					FOR CallRTBFL := 1 TO iRecipeBlockQty DO
						IF CallRTBFL > 0 AND CallRTBFL <= iRecipeBlockQty THEN
						AR2SiCalledRecipeTimeBlockNoCallArmTime[CallRTBFL, 1] :=	 AR3SiRecipeTimeBlockMemoryNoCallArmTime[iAutoModeCallRecipeTimeBlock_ProductRecipeNo, CallRTBFL, 1];
						AR2SiCalledRecipeTimeBlockNoCallArmTime[CallRTBFL, 2] :=	 AR3SiRecipeTimeBlockMemoryNoCallArmTime[iAutoModeCallRecipeTimeBlock_ProductRecipeNo, CallRTBFL, 2];
						AR2SiCalledRecipeTimeBlockNoCallArmTime[CallRTBFL, 3] :=	 AR3SiRecipeTimeBlockMemoryNoCallArmTime[iAutoModeCallRecipeTimeBlock_ProductRecipeNo, CallRTBFL, 3];
						AR2SiCalledRecipeTimeBlockNoCallArmTime[CallRTBFL, 4] :=	 AR3SiRecipeTimeBlockMemoryNoCallArmTime[iAutoModeCallRecipeTimeBlock_ProductRecipeNo, CallRTBFL, 4];
						AR2SiCalledRecipeTimeBlockNoCallArmTime[CallRTBFL, 5] :=	 AR3SiRecipeTimeBlockMemoryNoCallArmTime[iAutoModeCallRecipeTimeBlock_ProductRecipeNo, CallRTBFL, 5];
						AR2SiCalledRecipeTimeBlockNoCallArmTime[CallRTBFL, 6] :=	 AR3SiRecipeTimeBlockMemoryNoCallArmTime[iAutoModeCallRecipeTimeBlock_ProductRecipeNo, CallRTBFL, 6];
						AR2SiCalledRecipeTimeBlockNoCallArmTime[CallRTBFL, 7] :=	 AR3SiRecipeTimeBlockMemoryNoCallArmTime[iAutoModeCallRecipeTimeBlock_ProductRecipeNo, CallRTBFL, 7];
						AR2SiCalledRecipeTimeBlockNoCallArmTime[CallRTBFL, 8] :=	 AR3SiRecipeTimeBlockMemoryNoCallArmTime[iAutoModeCallRecipeTimeBlock_ProductRecipeNo, CallRTBFL, 8];
						AR2SiCalledRecipeTimeBlockNoCallArmTime[CallRTBFL, 9] :=	 AR3SiRecipeTimeBlockMemoryNoCallArmTime[iAutoModeCallRecipeTimeBlock_ProductRecipeNo, CallRTBFL, 9];
						END_IF
					END_FOR


				END_IF


				IF AR3SiRecipeTimeBlockMemoryWithCallArmTime[iAutoModeCallRecipeTimeBlock_ProductRecipeNo, 1, 3] <> 0 THEN
				CallRTBFL := 1;

					FOR CallRTBFL := 1 TO iRecipeBlockQty DO
						IF CallRTBFL > 0 AND CallRTBFL <= iRecipeBlockQty THEN
						AR2SiCalledRecipeTimeBlockWithCallArmTime[CallRTBFL, 1] :=	 AR3SiRecipeTimeBlockMemoryWithCallArmTime[iAutoModeCallRecipeTimeBlock_ProductRecipeNo, CallRTBFL, 1];
						AR2SiCalledRecipeTimeBlockWithCallArmTime[CallRTBFL, 2] :=	 AR3SiRecipeTimeBlockMemoryWithCallArmTime[iAutoModeCallRecipeTimeBlock_ProductRecipeNo, CallRTBFL, 2];
						AR2SiCalledRecipeTimeBlockWithCallArmTime[CallRTBFL, 3] :=	 AR3SiRecipeTimeBlockMemoryWithCallArmTime[iAutoModeCallRecipeTimeBlock_ProductRecipeNo, CallRTBFL, 3];
						AR2SiCalledRecipeTimeBlockWithCallArmTime[CallRTBFL, 4] :=	 AR3SiRecipeTimeBlockMemoryWithCallArmTime[iAutoModeCallRecipeTimeBlock_ProductRecipeNo, CallRTBFL, 4];
						AR2SiCalledRecipeTimeBlockWithCallArmTime[CallRTBFL, 5] :=	 AR3SiRecipeTimeBlockMemoryWithCallArmTime[iAutoModeCallRecipeTimeBlock_ProductRecipeNo, CallRTBFL, 5];
						AR2SiCalledRecipeTimeBlockWithCallArmTime[CallRTBFL, 6] :=	 AR3SiRecipeTimeBlockMemoryWithCallArmTime[iAutoModeCallRecipeTimeBlock_ProductRecipeNo, CallRTBFL, 6];
						AR2SiCalledRecipeTimeBlockWithCallArmTime[CallRTBFL, 7] :=	 AR3SiRecipeTimeBlockMemoryWithCallArmTime[iAutoModeCallRecipeTimeBlock_ProductRecipeNo, CallRTBFL, 7];
						AR2SiCalledRecipeTimeBlockWithCallArmTime[CallRTBFL, 8] :=	 AR3SiRecipeTimeBlockMemoryWithCallArmTime[iAutoModeCallRecipeTimeBlock_ProductRecipeNo, CallRTBFL, 8];
						AR2SiCalledRecipeTimeBlockWithCallArmTime[CallRTBFL, 9] :=	 AR3SiRecipeTimeBlockMemoryWithCallArmTime[iAutoModeCallRecipeTimeBlock_ProductRecipeNo, CallRTBFL, 9];
						END_IF
					END_FOR
			
			
				END_IF

			ELSE
			bInvalidCallRecipeTimeBlockNo := TRUE;
			END_IF

			IF AR2SiCalledRecipeTimeBlockWithCallArmTime [1,3] <> 0 THEN
			bCallRTB_NoTrackerInfo := FALSE;
			bCallRTB_CallOK := TRUE;
			END_IF

(*SimulatorMode Call*)
ELSIF bSimulatorModeEn
AND NOT bMasterTimeBlockScanningEn
AND NOT tProductRecipeChangesFound.Q
AND NOT  bScanningEN
AND iSimulatorModeCallRecipeTimeBlock_ProductRecipeNo >0
(*AND ARbProductRecipeTimeBlockAvailable[iSimulatorModeCallRecipeTimeBlock_ProductRecipeNo]
AND AR2SiCalledRecipeTimeBlockNoCallArmTime[1, 3] = 0*)
THEN

			IF iSimulatorModeCallRecipeTimeBlock_ProductRecipeNo >0 THEN
			AR2SiCalledRecipeTimeBlockNoCallArmTime := AR2SiCalledRecipeTimeBlockNoCallArmTimeEmpty;
			AR2SiCalledRecipeTimeBlockWithCallArmTime := AR2SiCalledRecipeTimeBlockWithCallArmTimeEmpty;
			bInvalidCallRecipeTimeBlockNo := FALSE;

				IF AR3SiRecipeTimeBlockMemoryNoCallArmTime[iSimulatorModeCallRecipeTimeBlock_ProductRecipeNo, 1, 3] <> 0 THEN
				CallRTBFL := 1;

					FOR CallRTBFL := 1 TO iRecipeBlockQty DO
						IF CallRTBFL > 0 AND CallRTBFL <= iRecipeBlockQty THEN
						AR2SiCalledRecipeTimeBlockNoCallArmTime[CallRTBFL, 1] :=	 AR3SiRecipeTimeBlockMemoryNoCallArmTime[iSimulatorModeCallRecipeTimeBlock_ProductRecipeNo, CallRTBFL, 1];
						AR2SiCalledRecipeTimeBlockNoCallArmTime[CallRTBFL, 2] :=	 AR3SiRecipeTimeBlockMemoryNoCallArmTime[iSimulatorModeCallRecipeTimeBlock_ProductRecipeNo, CallRTBFL, 2];
						AR2SiCalledRecipeTimeBlockNoCallArmTime[CallRTBFL, 3] :=	 AR3SiRecipeTimeBlockMemoryNoCallArmTime[iSimulatorModeCallRecipeTimeBlock_ProductRecipeNo, CallRTBFL, 3];
						AR2SiCalledRecipeTimeBlockNoCallArmTime[CallRTBFL, 4] :=	 AR3SiRecipeTimeBlockMemoryNoCallArmTime[iSimulatorModeCallRecipeTimeBlock_ProductRecipeNo, CallRTBFL, 4];
						AR2SiCalledRecipeTimeBlockNoCallArmTime[CallRTBFL, 5] :=	 AR3SiRecipeTimeBlockMemoryNoCallArmTime[iSimulatorModeCallRecipeTimeBlock_ProductRecipeNo, CallRTBFL, 5];
						AR2SiCalledRecipeTimeBlockNoCallArmTime[CallRTBFL, 6] :=	 AR3SiRecipeTimeBlockMemoryNoCallArmTime[iSimulatorModeCallRecipeTimeBlock_ProductRecipeNo, CallRTBFL, 6];
						AR2SiCalledRecipeTimeBlockNoCallArmTime[CallRTBFL, 7] :=	 AR3SiRecipeTimeBlockMemoryNoCallArmTime[iSimulatorModeCallRecipeTimeBlock_ProductRecipeNo, CallRTBFL, 7];
						AR2SiCalledRecipeTimeBlockNoCallArmTime[CallRTBFL, 8] :=	 AR3SiRecipeTimeBlockMemoryNoCallArmTime[iSimulatorModeCallRecipeTimeBlock_ProductRecipeNo, CallRTBFL, 8];
						AR2SiCalledRecipeTimeBlockNoCallArmTime[CallRTBFL, 9] :=	 AR3SiRecipeTimeBlockMemoryNoCallArmTime[iSimulatorModeCallRecipeTimeBlock_ProductRecipeNo, CallRTBFL, 9];
						END_IF
					END_FOR
			
			
				END_IF


				IF AR3SiRecipeTimeBlockMemoryWithCallArmTime[iSimulatorModeCallRecipeTimeBlock_ProductRecipeNo, 1, 3] <> 0 THEN
				CallRTBFL := 1;
			
					FOR CallRTBFL := 1 TO iRecipeBlockQty DO
						IF CallRTBFL > 0 AND CallRTBFL <= iRecipeBlockQty THEN
						AR2SiCalledRecipeTimeBlockWithCallArmTime[CallRTBFL, 1] :=	 AR3SiRecipeTimeBlockMemoryWithCallArmTime[iSimulatorModeCallRecipeTimeBlock_ProductRecipeNo, CallRTBFL, 1];
						AR2SiCalledRecipeTimeBlockWithCallArmTime[CallRTBFL, 2] :=	 AR3SiRecipeTimeBlockMemoryWithCallArmTime[iSimulatorModeCallRecipeTimeBlock_ProductRecipeNo, CallRTBFL, 2];
						AR2SiCalledRecipeTimeBlockWithCallArmTime[CallRTBFL, 3] :=	 AR3SiRecipeTimeBlockMemoryWithCallArmTime[iSimulatorModeCallRecipeTimeBlock_ProductRecipeNo, CallRTBFL, 3];
						AR2SiCalledRecipeTimeBlockWithCallArmTime[CallRTBFL, 4] :=	 AR3SiRecipeTimeBlockMemoryWithCallArmTime[iSimulatorModeCallRecipeTimeBlock_ProductRecipeNo, CallRTBFL, 4];
						AR2SiCalledRecipeTimeBlockWithCallArmTime[CallRTBFL, 5] :=	 AR3SiRecipeTimeBlockMemoryWithCallArmTime[iSimulatorModeCallRecipeTimeBlock_ProductRecipeNo, CallRTBFL, 5];
						AR2SiCalledRecipeTimeBlockWithCallArmTime[CallRTBFL, 6] :=	 AR3SiRecipeTimeBlockMemoryWithCallArmTime[iSimulatorModeCallRecipeTimeBlock_ProductRecipeNo, CallRTBFL, 6];
						AR2SiCalledRecipeTimeBlockWithCallArmTime[CallRTBFL, 7] :=	 AR3SiRecipeTimeBlockMemoryWithCallArmTime[iSimulatorModeCallRecipeTimeBlock_ProductRecipeNo, CallRTBFL, 7];
						AR2SiCalledRecipeTimeBlockWithCallArmTime[CallRTBFL, 8] :=	 AR3SiRecipeTimeBlockMemoryWithCallArmTime[iSimulatorModeCallRecipeTimeBlock_ProductRecipeNo, CallRTBFL, 8];
						AR2SiCalledRecipeTimeBlockWithCallArmTime[CallRTBFL, 9] :=	 AR3SiRecipeTimeBlockMemoryWithCallArmTime[iSimulatorModeCallRecipeTimeBlock_ProductRecipeNo, CallRTBFL, 9];
						END_IF
					END_FOR

			
				END_IF

			ELSE
			bInvalidCallRecipeTimeBlockNo := TRUE;
			END_IF


			IF AR2SiCalledRecipeTimeBlockWithCallArmTime [1,3] <> 0 THEN
			bCallRTB_NoTrackerInfo := FALSE;
			bCallRTB_CallOK := TRUE;
			END_IF


END_IF



(*Check Product Recipe Time Block Availibility *)
iCheckPRTBFL := 1;

	FOR iCheckPRTBFL := 1 TO iProductRecipeArrayQty DO
		IF iCheckPRTBFL >= 1 AND iCheckPRTBFL <= iProductRecipeArrayQty THEN

			IF  AR3SiRecipeTimeBlockMemoryNoCallArmTime[iCheckPRTBFL, 1, 3] > 0 THEN
			ARbProductRecipeTimeBlockAvailable[iCheckPRTBFL ] := TRUE;
			ELSE
			ARbProductRecipeTimeBlockAvailable[iCheckPRTBFL ] := FALSE;
			END_IF

		END_IF
	END_FOR

ACTION XML_ImportExport:
(* XML Import Export Control *)
(*	ARiSubAction					: ARRAY [1..10] OF INT; (* 0-Idle, 1-Import, 2-Export, 3-Clear/Delete 8-Done *)*)

	IF 		ARiSubAction[2] = 1 THEN (*Write from Buffer to Actual Memory*)

				CallRTBFL := 1;

					FOR CallRTBFL := 1 TO iRecipeBlockQty DO
						IF CallRTBFL > 0 AND CallRTBFL <= iRecipeBlockQty THEN
						AR3SiRecipeTimeBlockMemoryNoCallArmTime[iXMLRecipeNo, CallRTBFL, 1] :=	 DSV3XML_Recipe.AR2SiRecipeTimeBlockNoCallArmTime[CallRTBFL, 1];
						AR3SiRecipeTimeBlockMemoryNoCallArmTime[iXMLRecipeNo, CallRTBFL, 2] :=	 DSV3XML_Recipe.AR2SiRecipeTimeBlockNoCallArmTime[CallRTBFL, 2];
						AR3SiRecipeTimeBlockMemoryNoCallArmTime[iXMLRecipeNo, CallRTBFL, 3] :=	 DSV3XML_Recipe.AR2SiRecipeTimeBlockNoCallArmTime[CallRTBFL, 3];
						AR3SiRecipeTimeBlockMemoryNoCallArmTime[iXMLRecipeNo, CallRTBFL, 4] :=	 DSV3XML_Recipe.AR2SiRecipeTimeBlockNoCallArmTime[CallRTBFL, 4];
						AR3SiRecipeTimeBlockMemoryNoCallArmTime[iXMLRecipeNo, CallRTBFL, 5] :=	 DSV3XML_Recipe.AR2SiRecipeTimeBlockNoCallArmTime[CallRTBFL, 5];
						AR3SiRecipeTimeBlockMemoryNoCallArmTime[iXMLRecipeNo, CallRTBFL, 6] :=	 DSV3XML_Recipe.AR2SiRecipeTimeBlockNoCallArmTime[CallRTBFL, 6];
						AR3SiRecipeTimeBlockMemoryNoCallArmTime[iXMLRecipeNo, CallRTBFL, 7] :=	 DSV3XML_Recipe.AR2SiRecipeTimeBlockNoCallArmTime[CallRTBFL, 7];
						AR3SiRecipeTimeBlockMemoryNoCallArmTime[iXMLRecipeNo, CallRTBFL, 8] :=	 DSV3XML_Recipe.AR2SiRecipeTimeBlockNoCallArmTime[CallRTBFL, 8];
						AR3SiRecipeTimeBlockMemoryNoCallArmTime[iXMLRecipeNo, CallRTBFL, 9] :=	 DSV3XML_Recipe.AR2SiRecipeTimeBlockNoCallArmTime[CallRTBFL, 9];

						AR3SiRecipeTimeBlockMemoryWithCallArmTime[iXMLRecipeNo, CallRTBFL, 1] :=	 DSV3XML_Recipe.AR2SiRecipeTimeBlockWithCallArmTime[CallRTBFL, 1];
						AR3SiRecipeTimeBlockMemoryWithCallArmTime[iXMLRecipeNo, CallRTBFL, 2] :=	 DSV3XML_Recipe.AR2SiRecipeTimeBlockWithCallArmTime[CallRTBFL, 2];
						AR3SiRecipeTimeBlockMemoryWithCallArmTime[iXMLRecipeNo, CallRTBFL, 3] :=	 DSV3XML_Recipe.AR2SiRecipeTimeBlockWithCallArmTime[CallRTBFL, 3];
						AR3SiRecipeTimeBlockMemoryWithCallArmTime[iXMLRecipeNo, CallRTBFL, 4] :=	 DSV3XML_Recipe.AR2SiRecipeTimeBlockWithCallArmTime[CallRTBFL, 4];
						AR3SiRecipeTimeBlockMemoryWithCallArmTime[iXMLRecipeNo, CallRTBFL, 5] :=	 DSV3XML_Recipe.AR2SiRecipeTimeBlockWithCallArmTime[CallRTBFL, 5];
						AR3SiRecipeTimeBlockMemoryWithCallArmTime[iXMLRecipeNo, CallRTBFL, 6] :=	 DSV3XML_Recipe.AR2SiRecipeTimeBlockWithCallArmTime[CallRTBFL, 6];
						AR3SiRecipeTimeBlockMemoryWithCallArmTime[iXMLRecipeNo, CallRTBFL, 7] :=	 DSV3XML_Recipe.AR2SiRecipeTimeBlockWithCallArmTime[CallRTBFL, 7];
						AR3SiRecipeTimeBlockMemoryWithCallArmTime[iXMLRecipeNo, CallRTBFL, 8] :=	 DSV3XML_Recipe.AR2SiRecipeTimeBlockWithCallArmTime[CallRTBFL, 8];
						AR3SiRecipeTimeBlockMemoryWithCallArmTime[iXMLRecipeNo, CallRTBFL, 9] :=	 DSV3XML_Recipe.AR2SiRecipeTimeBlockWithCallArmTime[CallRTBFL, 9];
						END_IF
					END_FOR

				ARbProductRecipeTimeBlockAvailable[iXMLRecipeNo] := DSV3XML_Recipe.bProductRecipeTimeBlockAvailable ;

				ARiSubAction[2] := 8;
(*				IF iHMIRecipeNo = iXMLRecipeNo THEN
					bRecipeLoadPb := TRUE;
				END_IF
*)
	ELSIF	ARiSubAction[2] = 2 THEN (*Read from Actual to Buffer Memory*)

				CallRTBFL := 1;

					FOR CallRTBFL := 1 TO iRecipeBlockQty DO
						IF CallRTBFL > 0 AND CallRTBFL <= iRecipeBlockQty THEN
						DSV3XML_Recipe.AR2SiRecipeTimeBlockNoCallArmTime[CallRTBFL, 1] :=	 AR3SiRecipeTimeBlockMemoryNoCallArmTime[iXMLRecipeNo, CallRTBFL, 1];
						DSV3XML_Recipe.AR2SiRecipeTimeBlockNoCallArmTime[CallRTBFL, 2] :=	 AR3SiRecipeTimeBlockMemoryNoCallArmTime[iXMLRecipeNo, CallRTBFL, 2];
						DSV3XML_Recipe.AR2SiRecipeTimeBlockNoCallArmTime[CallRTBFL, 3] :=	 AR3SiRecipeTimeBlockMemoryNoCallArmTime[iXMLRecipeNo, CallRTBFL, 3];
						DSV3XML_Recipe.AR2SiRecipeTimeBlockNoCallArmTime[CallRTBFL, 4] :=	 AR3SiRecipeTimeBlockMemoryNoCallArmTime[iXMLRecipeNo, CallRTBFL, 4];
						DSV3XML_Recipe.AR2SiRecipeTimeBlockNoCallArmTime[CallRTBFL, 5] :=	 AR3SiRecipeTimeBlockMemoryNoCallArmTime[iXMLRecipeNo, CallRTBFL, 5];
						DSV3XML_Recipe.AR2SiRecipeTimeBlockNoCallArmTime[CallRTBFL, 6] :=	 AR3SiRecipeTimeBlockMemoryNoCallArmTime[iXMLRecipeNo, CallRTBFL, 6];
						DSV3XML_Recipe.AR2SiRecipeTimeBlockNoCallArmTime[CallRTBFL, 7] :=	 AR3SiRecipeTimeBlockMemoryNoCallArmTime[iXMLRecipeNo, CallRTBFL, 7];
						DSV3XML_Recipe.AR2SiRecipeTimeBlockNoCallArmTime[CallRTBFL, 8] :=	 AR3SiRecipeTimeBlockMemoryNoCallArmTime[iXMLRecipeNo, CallRTBFL, 8];
						DSV3XML_Recipe.AR2SiRecipeTimeBlockNoCallArmTime[CallRTBFL, 9] :=	 AR3SiRecipeTimeBlockMemoryNoCallArmTime[iXMLRecipeNo, CallRTBFL, 9];

						DSV3XML_Recipe.AR2SiRecipeTimeBlockWithCallArmTime[CallRTBFL, 1] :=	 AR3SiRecipeTimeBlockMemoryWithCallArmTime[iXMLRecipeNo, CallRTBFL, 1];
						DSV3XML_Recipe.AR2SiRecipeTimeBlockWithCallArmTime[CallRTBFL, 2] :=	 AR3SiRecipeTimeBlockMemoryWithCallArmTime[iXMLRecipeNo, CallRTBFL, 2];
						DSV3XML_Recipe.AR2SiRecipeTimeBlockWithCallArmTime[CallRTBFL, 3] :=	 AR3SiRecipeTimeBlockMemoryWithCallArmTime[iXMLRecipeNo, CallRTBFL, 3];
						DSV3XML_Recipe.AR2SiRecipeTimeBlockWithCallArmTime[CallRTBFL, 4] :=	 AR3SiRecipeTimeBlockMemoryWithCallArmTime[iXMLRecipeNo, CallRTBFL, 4];
						DSV3XML_Recipe.AR2SiRecipeTimeBlockWithCallArmTime[CallRTBFL, 5] :=	 AR3SiRecipeTimeBlockMemoryWithCallArmTime[iXMLRecipeNo, CallRTBFL, 5];
						DSV3XML_Recipe.AR2SiRecipeTimeBlockWithCallArmTime[CallRTBFL, 6] :=	 AR3SiRecipeTimeBlockMemoryWithCallArmTime[iXMLRecipeNo, CallRTBFL, 6];
						DSV3XML_Recipe.AR2SiRecipeTimeBlockWithCallArmTime[CallRTBFL, 7] :=	 AR3SiRecipeTimeBlockMemoryWithCallArmTime[iXMLRecipeNo, CallRTBFL, 7];
						DSV3XML_Recipe.AR2SiRecipeTimeBlockWithCallArmTime[CallRTBFL, 8] :=	 AR3SiRecipeTimeBlockMemoryWithCallArmTime[iXMLRecipeNo, CallRTBFL, 8];
						DSV3XML_Recipe.AR2SiRecipeTimeBlockWithCallArmTime[CallRTBFL, 9] :=	 AR3SiRecipeTimeBlockMemoryWithCallArmTime[iXMLRecipeNo, CallRTBFL, 9];
						END_IF
					END_FOR

				DSV3XML_Recipe.bProductRecipeTimeBlockAvailable := ARbProductRecipeTimeBlockAvailable[iXMLRecipeNo];

				ARiSubAction[2] := 8;

	ELSIF	ARiSubAction[2] = 3 THEN (*DELETE Actual Memory*)

				AR3SiRecipeTimeBlockMemoryNoCallArmTime		:= AR3SiRecipeTimeBlockMemoryNoCallArmTime_Delete;
				AR3SiRecipeTimeBlockMemoryWithCallArmTime 		:= AR3SiRecipeTimeBlockMemoryWithCallArmTime_Delete;
				ARbProductRecipeTimeBlockAvailable 				:= ARbProductRecipeTimeBlockAvailable_Delete;

				ARiSubAction[2] := 8;
(*				IF iHMIRecipeNo = iXMLRecipeNo THEN
					bRecipeLoadPb := TRUE;
				END_IF
*)
	END_IF
END_ACTION

END_FUNCTION_BLOCK

// ---- FBs/B_JKS_NewFB_V3/UserCtrl/FB3_HmiTF1800_UserlevelManagement.TcPOU
FUNCTION_BLOCK FB3_HmiTF1800_UserlevelManagement
VAR_INPUT
	
	bLoginPB 					: BOOL;
	bLogoutPB 					: BOOL;
	iLoginNameId 				: REFERENCE TO INT; // The LoginName selection in HMI during User Login Pop-up Screen, the choosen user will translated as Array ID No and pass here.
	sPasswordField 				: REFERENCE TO STRING; // Similar to Var In/Out so that i can clear the password if login failed
	
	iUM_SelectedLoginNameId	 	: REFERENCE TO INT;		// User Management - Selected Login Name ID (Array No)

	sUM_CurrentPassword			: REFERENCE TO STRING;	// User Management - Current Password (For password change only)
	sUM_NewPassword				: REFERENCE TO STRING;	// User Management - New Password (For password change or new user registration)
	sUM_ConfirmPassword			: REFERENCE TO STRING;	// User Management - New Password (For password change or new user registration)

	sUM_NewUserLoginName		: REFERENCE TO STRING;	// User Management - New User Login Name
	sUM_NewUserGroupId			: REFERENCE TO INT;		// User Management - Select from UserGroupList

	sUM_NewUserOperatorIdentifier	: REFERENCE TO STRING;
	sUM_NewUserActorType			: REFERENCE TO eActor;
	sUM_NewUserLastName				: REFERENCE TO STRING;
	sUM_NewUserFirstName			: REFERENCE TO STRING;
//	sUM_NewUserGroupName			: REFERENCE TO WSTRING; // Generated by reference eto sUM_NewUserGroupId
	
	bUM_CreatePB				: BOOL;		// User Management - Button for New User creation
	bUM_EditPB					: BOOL;		// User Management - Button for Edit User
	bUM_DeletePB				: BOOL;		// User Management - Button for Delete User
	bUM_EnablePB				: BOOL; 	// to Enable selected User
	bUM_DisablePB				: BOOL; 	// to Temporary Disable selected User
	bUM_ConfirmPB				: BOOL;		// for Edit, Delete and Disable used. click to save
	bUM_ReturnPB				: BOOL;		// for Edit, Delete and Disable used, click to return without save.
		
END_VAR
VAR_OUTPUT
	dsHmiUserStatus_Active		: DS_HmiUserStatus;
	dsHmiUserStatus_Login		: DS_HmiUserStatus;
	dsHmiUserStatus_Logout		: DS_HmiUserStatus;
	
//	iActiveUserGroupId			: INT;
//	sActiveLoginName			: STRING;
	
//	sActiveOperatorIdentifier	: STRING;
//	eActiveActorType			: eActor;
//	sActiveLastName				: STRING;
//	sActiveFirstName			: STRING;
	wsActiveUserGroupName		: WSTRING;
	sMessage					: STRING;
	
END_VAR
VAR
	tsLocalSystemTimeStruct		: TIMESTRUCT;
	dsHmiUserStatus_Empty		: DS_HmiUserStatus;

	ARsUserGroup 				: ARRAY [0..5] OF WSTRING;	// Default UserGroup - Must Matched with HMI UserGroup Naming
	
	bLoginPBRE		: R_TRIG;
	bLogoutPBRE		: R_TRIG;
	bUM_CreatePBRE	: R_TRIG;
	bUM_EditPBRE	: R_TRIG;
	bUM_DeletePBRE	: R_TRIG;
	bUM_DisablePBRE	: R_TRIG;
	iCase: INT;
	sMessageDelayTimer: TON;
	iFL: INT;
	bDuplicatedLoginName: BOOL;
	bDuplicatedOperatorId: BOOL;
	bUserDBMax: BOOL;
	iUserDBVacantField: INT;
	bUM_ConfirmPBRE: R_TRIG;
	bUM_ReturnPBRE: R_TRIG;
	btest: BOOL;
	bUM_EnablePBRE: R_TRIG;
	tLoginActivatedTimer: TON;
	tLogoutActivatedTimer: TON;
	ntGetTime: NT_GetTime;
	t1s: TON;
END_VAR
	
VAR PERSISTENT
	dsHmiUserReg 			: DS_HmiUserReg;
END_VAR

t1s(IN:=NOT t1s.Q , PT:=T#0.5S , Q=> , ET=> );

// Get System Time
ntGetTime(	NETID:='' , START:=t1s.Q , TMOUT:= T#5S, TIMESTR=> tsLocalSystemTimeStruct);

tsLocalSystemTimeStruct.wYear;
tsLocalSystemTimeStruct.wMonth;
tsLocalSystemTimeStruct.wDay;
tsLocalSystemTimeStruct.wHour;
tsLocalSystemTimeStruct.wMinute;
tsLocalSystemTimeStruct.wSecond;
tsLocalSystemTimeStruct.wMilliseconds;
tsLocalSystemTimeStruct.wDayOfWeek;


// Default UserGroup - Must Matched with HMI UserGroup Naming
ARsUserGroup[0]			:= 	STRING_TO_WSTRING('GUEST');
ARsUserGroup[1]			:= 	STRING_TO_WSTRING('OPERATOR');
ARsUserGroup[2]			:=	STRING_TO_WSTRING('TECHNICIAN');
ARsUserGroup[3]			:=	STRING_TO_WSTRING('ENGINEER');
ARsUserGroup[4]			:=	STRING_TO_WSTRING('ADMIN');
ARsUserGroup[5]			:=	STRING_TO_WSTRING('JKS');
//ARsUserGroup[6]			:=	STRING_TO_WSTRING('');
//ARsUserGroup[7]			:=	STRING_TO_WSTRING('');	

// Default SuperAdmin
dsHmiUserReg.ARbUserStatus[dsHmiUserReg.iQtyUserReg+1]			:= 	TRUE		;
dsHmiUserReg.AReActorType[dsHmiUserReg.iQtyUserReg+1]			:= 	0			; //Human
dsHmiUserReg.ARiUserGroupID[dsHmiUserReg.iQtyUserReg+1]			:= 	5			; //Highest level - JKS Admin
dsHmiUserReg.ARsFirstName[dsHmiUserReg.iQtyUserReg+1]			:= 	'Machine'	;
dsHmiUserReg.ARsLastName[dsHmiUserReg.iQtyUserReg+1]			:= 	'Maker'		;
dsHmiUserReg.ARsLoginName[dsHmiUserReg.iQtyUserReg+1]			:= 	'SoftwareManager'	;
dsHmiUserReg.ARsOperatorIdentifier[dsHmiUserReg.iQtyUserReg+1]	:= 	'Software Manager'	;
dsHmiUserReg.ARsPw[dsHmiUserReg.iQtyUserReg+1]					:= 	'7189'	;
dsHmiUserReg.ARwsUserGroupName[dsHmiUserReg.iQtyUserReg+1]		:= 	ARsUserGroup[5]	;


// R_TRIG
bLoginPBRE		(CLK:=bLoginPB , 		Q=> );
bLogoutPBRE		(CLK:=bLogoutPB , 		Q=> );

bUM_CreatePBRE	(CLK:=bUM_CreatePB , 	Q=> );
bUM_EditPBRE	(CLK:=bUM_EditPB , 		Q=> );
bUM_DeletePBRE	(CLK:=bUM_DeletePB , 	Q=> );
bUM_EnablePBRE	(CLK:=bUM_EnablePB , 	Q=> );
bUM_DisablePBRE	(CLK:=bUM_DisablePB , 	Q=> );
bUM_ConfirmPBRE	(CLK:=bUM_ConfirmPB , 	Q=> );
bUM_ReturnPBRE	(CLK:=bUM_ReturnPB , 	Q=> );


// Delay off
tLoginActivatedTimer(IN:=dsHmiUserStatus_Login.bActivatedFlag , PT:=T#1S , Q=> , ET=> );
IF tLoginActivatedTimer.Q THEN
	dsHmiUserStatus_Login.bActivatedFlag := FALSE;
END_IF

tLogoutActivatedTimer(IN:=dsHmiUserStatus_Logout.bActivatedFlag , PT:=T#1S , Q=> , ET=> );
IF tLogoutActivatedTimer.Q THEN
	dsHmiUserStatus_Logout.bActivatedFlag := FALSE;
END_IF



// Action 

	IF iCase = 0 THEN
		
		IF 	bLoginPBRE.Q AND iLoginNameId > 0 AND iLoginNameId <= dsHmiUserReg.iQtyUserReg +1 AND sPasswordField <> '' THEN
			iCase := 11; // Login 
			
		ELSIF bLogoutPBRE.Q THEN
			iCase := 21; //	Logout
			
		ELSIF bUM_CreatePBRE.Q AND dsHmiUserStatus_Login.sUserGroupId >= 4 THEN
			iCase := 31; //	User Management -> New User Creation
			
		ELSIF bUM_EditPBRE.Q AND dsHmiUserStatus_Login.sUserGroupId >= 4 AND iUM_SelectedLoginNameId > 0 AND iUM_SelectedLoginNameId <= dsHmiUserReg.iQtyUserReg +1 THEN
			iCase := 41; //	User Management -> Edit User
			
		ELSIF bUM_DeletePBRE.Q AND dsHmiUserStatus_Login.sUserGroupId >= 4 AND iUM_SelectedLoginNameId > 0 AND iUM_SelectedLoginNameId <= dsHmiUserReg.iQtyUserReg +1 
		AND dsHmiUserReg.ARsLoginName[iUM_SelectedLoginNameId] <> dsHmiUserStatus_Login.sLoginName THEN
			iCase := 51; //	User Management -> Delete User
			
		ELSIF (bUM_EnablePBRE.Q OR bUM_DisablePBRE.Q)AND dsHmiUserStatus_Login.sUserGroupId >= 4 AND iUM_SelectedLoginNameId > 0 AND iUM_SelectedLoginNameId <= dsHmiUserReg.iQtyUserReg +1 THEN
			iCase := 61; //	User Management -> Enable or Temporary Disable selected User

		ELSIF (bUM_DeletePBRE.Q) AND dsHmiUserReg.ARsLoginName[iUM_SelectedLoginNameId] = dsHmiUserStatus_Login.sLoginName THEN
				sMessage := 'Signed in user cannot be delete, please sign in another administrator user before deletion';
					
		ELSIF (bUM_CreatePBRE.Q OR bUM_EditPBRE.Q OR bUM_DeletePBRE.Q OR bUM_EnablePBRE.Q OR bUM_DisablePBRE.Q ) AND dsHmiUserStatus_Login.sUserGroupId <= 4  THEN
				sMessage := 'You do not have permission to perform the task, please contact administrator.';
					
		ELSIF (bUM_EditPBRE.Q OR bUM_DeletePBRE.Q OR bUM_EnablePBRE.Q OR bUM_DisablePBRE.Q ) AND iUM_SelectedLoginNameId = 0 THEN
				sMessage := 'Please select user';
					
		ELSIF (bUM_EditPBRE.Q OR bUM_DeletePBRE.Q OR bUM_EnablePBRE.Q OR bUM_DisablePBRE.Q ) AND iUM_SelectedLoginNameId > dsHmiUserReg.iQtyUserReg +1 THEN
				sMessage := 'Selected user out of user database range';
					
		ELSIF bLoginPBRE.Q AND (iLoginNameId = 0 OR sPasswordField = '' ) THEN
				sMessage := 'Please select user and enter password to login';
					
		ELSIF bLoginPBRE.Q AND iLoginNameId > dsHmiUserReg.iQtyUserReg +1 THEN
				sMessage := 'Selected login user out of user database range';
					
		END_IF
		
	END_IF



CASE iCase OF
	
	0: ;// Idling;

	8: // Clear new user registration field and return

		sUM_CurrentPassword 			:= '' ;
		sUM_NewPassword 				:= '' ;
		sUM_ConfirmPassword 			:= '' ; 
		sUM_NewUserLoginName 			:= '' ; 
		sUM_NewUserGroupId				:= 0 ;	
		sUM_NewUserOperatorIdentifier	:= '' ;
		sUM_NewUserActorType			:= 0 ; 
		sUM_NewUserLastName				:= '' ;
		sUM_NewUserFirstName			:= '' ;
		
		iUM_SelectedLoginNameId			:= 0;
		
		iCase := 0; // Return		
	
	9: // Clear Active Field and return
	
		dsHmiUserStatus_Logout := dsHmiUserStatus_Active;
		IF dsHmiUserStatus_Logout.sLoginName <> '' THEN
			dsHmiUserStatus_Logout.bActivatedFlag 	:= TRUE;
			dsHmiUserStatus_Logout.tsDateTime 		:= tsLocalSystemTimeStruct;
		END_IF

		sPasswordField 			:= 		'';
		dsHmiUserStatus_Active 	:= 		dsHmiUserStatus_Empty;
		wsActiveUserGroupName 	:= 		TO_WSTRING('');

		iCase := 0; //Return



	11: // Login 
	
		IF dsHmiUserReg.ARsPw[iLoginNameId] = sPasswordField AND dsHmiUserReg.ARbUserStatus[iLoginNameId] THEN
				
				// if detected with existing login user and it relogin with another user, this section will action
				IF dsHmiUserStatus_Active.sLoginName <> '' THEN
					dsHmiUserStatus_Logout := dsHmiUserStatus_Active;
					dsHmiUserStatus_Logout.bActivatedFlag := TRUE;
					dsHmiUserStatus_Logout.tsDateTime := tsLocalSystemTimeStruct;
				END_IF


				sPasswordField 				:= 		'';
				
				dsHmiUserStatus_Active.bActivatedFlag		:= 		TRUE;
				dsHmiUserStatus_Active.sOperatorIdentifier 	:= 		dsHmiUserReg.ARsOperatorIdentifier[iLoginNameId];	// Celestica Requirement
				dsHmiUserStatus_Active.eActorType			:=		dsHmiUserReg.AReActorType[iLoginNameId];			// Celestica Requirement
				dsHmiUserStatus_Active.sULastName			:=		dsHmiUserReg.ARsLastName[iLoginNameId];
				dsHmiUserStatus_Active.sFirstName			:=		dsHmiUserReg.ARsFirstName[iLoginNameId];
				
				dsHmiUserStatus_Active.sLoginName			:=		dsHmiUserReg.ARsLoginName[iLoginNameId];			// Same as Username
	
				dsHmiUserStatus_Active.sUserGroupId			:=		dsHmiUserReg.ARiUserGroupID[iLoginNameId];			// Define in HMI TF1800

				dsHmiUserStatus_Active.tsDateTime			:=		tsLocalSystemTimeStruct;
				wsActiveUserGroupName 						:= 		dsHmiUserReg.ARwsUserGroupName[iLoginNameId];
				
	
				dsHmiUserStatus_Login := dsHmiUserStatus_Active;
				dsHmiUserStatus_Login.bActivatedFlag := TRUE;
				dsHmiUserStatus_Login.tsDateTime := tsLocalSystemTimeStruct;
				
				sMessage := 'Welcome!';
				sMessage := concat(sMessage,' ');
				sMessage := concat(sMessage,dsHmiUserStatus_Active.sFirstName);
				sMessage := concat(sMessage,' ');
				sMessage := concat(sMessage,dsHmiUserStatus_Active.sULastName);
				sMessage := concat(sMessage,' (');
				sMessage := concat(sMessage,dsHmiUserStatus_Active.sLoginName);
				sMessage := concat(sMessage,')');
		
				iCase := 0;	//Return
						
		ELSIF NOT dsHmiUserReg.ARbUserStatus[iLoginNameId] THEN
				sMessage := 'Selected user has been DISABLE, please contact administrator.';
				iCase := 9; // Clear Active Field and return
			
		
		ELSE
				sMessage := 'Invalid password';
				iCase := 9; // Clear Active Field and return
		
		END_IF
				
		
	
	21: // Logout 
		
				sMessage := 'You have been successfully logged out.';	
				iCase := 9; // Clear Active Field and return 
		
	
	31: // User Management -> New User Creation 
	
		IF sUM_NewPassword 					<> '' 
		AND sUM_ConfirmPassword 			<> '' 
	//	AND sUM_NewUserLoginName 			<> '' 
		AND sUM_NewUserGroupId				<> 0 AND sUM_NewUserGroupId <= 4	// Doesnt need for another JKS User (5)
	//	AND sUM_NewUserOperatorIdentifier	<> ''
	//	AND sUM_NewUserActorType			<= 2 AND sUM_NewUserActorType >= 0
		AND sUM_NewUserLastName				<> ''
		AND sUM_NewUserFirstName			<> ''

		THEN
			
			// Check Duplicated Login Name
				bDuplicatedLoginName := FALSE;
				
				FOR iFL := 1 TO dsHmiUserReg.iQtyUserReg DO
					IF sUM_NewUserLoginName = dsHmiUserReg.ARsLoginName[iFL] THEN
						bDuplicatedLoginName := TRUE;
						EXIT;
					END_IF
				;
				END_FOR

			// Check Duplicated Operator Identifier
				bDuplicatedOperatorId := FALSE;
				
				FOR iFL := 1 TO dsHmiUserReg.iQtyUserReg DO
					IF sUM_NewUserOperatorIdentifier = dsHmiUserReg.ARsOperatorIdentifier[iFL] THEN
						bDuplicatedOperatorId := TRUE;
						EXIT;
					END_IF
				;
				END_FOR

			// Check User Database Limit
				bUserDBMax := TRUE;
				iUserDBVacantField := 0;
				
				FOR iFL := 1 TO dsHmiUserReg.iQtyUserReg DO
					IF dsHmiUserReg.ARsLoginName[iFL] = '' THEN
						iUserDBVacantField := iFL;
						bUserDBMax := FALSE;
						EXIT;
					END_IF
				;
				END_FOR


			IF sUM_NewPassword <> sUM_ConfirmPassword THEN
				
				sMessage := 'Your new password and confirmation password mismatched';	
				sUM_ConfirmPassword := '';
				iCase := 0;

			ELSIF bDuplicatedLoginName THEN
							
				sMessage := 'Login Name already exists, please try with another one ';	
				sUM_NewUserLoginName 	:= '';
				sUM_NewPassword			:= '';
				sUM_ConfirmPassword 	:= '';
				iCase 					:= 0;

//			ELSIF bDuplicatedOperatorId THEN
							
//				sMessage := 'Operator Indentifier already exists, please try with another one ';	
//				sUM_NewUserOperatorIdentifier 	:= '';
//				sUM_NewPassword					:= '';
//				sUM_ConfirmPassword 			:= '';
//				iCase 							:= 0;
				
			ELSIF bUserDBMax THEN
							
				sMessage 	:= 'User Registration Limit Reached. Please delete at least one user to proceed the registration again ';	
				iCase 		:= 8; // Clear new user registration field and return
				
			ELSE
				
				
							
			//	dsHmiUserReg.ARsOperatorIdentifier[iUserDBVacantField] 	:= sUM_NewUserOperatorIdentifier;	// Celestica Requirement
			//	dsHmiUserReg.AReActorType[iUserDBVacantField]			:= sUM_NewUserActorType;			// Celestica Requirement
				dsHmiUserReg.ARsLastName[iUserDBVacantField]			:= sUM_NewUserLastName;
				dsHmiUserReg.ARsFirstName[iUserDBVacantField]			:= sUM_NewUserFirstName;
				dsHmiUserReg.ARsLoginName[iUserDBVacantField]			:= sUM_NewUserLoginName;			// Same as Username
				dsHmiUserReg.ARbUserStatus[iUserDBVacantField]			:= TRUE;							// 0 = Deactivated/Disable, 1 = Active User
				
				dsHmiUserReg.ARiUserGroupID[iUserDBVacantField]			:= sUM_NewUserGroupId;				// Define in HMI TF1800
				dsHmiUserReg.ARwsUserGroupName[iUserDBVacantField]		:= ARsUserGroup[sUM_NewUserGroupId];// Define in HMI TF1800
				dsHmiUserReg.ARsPw[iUserDBVacantField]					:= sUM_NewPassword;		

				sMessage := 'User is added successfully. Please go to Login page to proceed';	
				iCase := 8; // Clear new user registration field and return
					
			END_IF
			
		
		ELSE
			
			sMessage := 'Your registration is Incomplete';	
			iCase := 0; //RETURN
		END_IF
	
		
	41: // User Management -> Edit User 

		sUM_NewUserOperatorIdentifier := dsHmiUserReg.ARsOperatorIdentifier[iUM_SelectedLoginNameId];	// Celestica Requirement
		sUM_NewUserActorType := dsHmiUserReg.AReActorType[iUM_SelectedLoginNameId];						// Celestica Requirement
		sUM_NewUserLastName := dsHmiUserReg.ARsLastName[iUM_SelectedLoginNameId];
		sUM_NewUserFirstName := dsHmiUserReg.ARsFirstName[iUM_SelectedLoginNameId];
		sUM_NewUserLoginName := dsHmiUserReg.ARsLoginName[iUM_SelectedLoginNameId];						// Same as Username
		
		sUM_NewUserGroupId := dsHmiUserReg.ARiUserGroupID[iUM_SelectedLoginNameId];						// Define in HMI TF1800

		sUM_CurrentPassword := '';//dsHmiUserReg.ARsPw[iUM_SelectedLoginNameId];		
		sUM_NewPassword 	:= '';//dsHmiUserReg.ARsPw[iUM_SelectedLoginNameId];		
		sUM_ConfirmPassword := '';//dsHmiUserReg.ARsPw[iUM_SelectedLoginNameId];		
		
		iCase := 42;

	42: // User Management -> Edit User => Waiting Confirmation
	
		sMessage := 'Are you sure you want to MODIFY selected user?';	
	
		IF bUM_ConfirmPBRE.Q THEN
					
			IF sUM_CurrentPassword <> dsHmiUserReg.ARsPw[iUM_SelectedLoginNameId] THEN
					
				sMessage := 'Invalid Current Password';
				iUM_SelectedLoginNameId := 0;	
				iCase := 8; // Clear and return
			
			ELSIF sUM_NewPassword <> sUM_ConfirmPassword THEN	
			
					
				sMessage := 'Your new password and confirmation password mismatched';
				iUM_SelectedLoginNameId := 0;	
				iCase := 8; // Clear and return
			
			ELSE
				dsHmiUserReg.ARsOperatorIdentifier[iUM_SelectedLoginNameId] 	:= sUM_NewUserOperatorIdentifier;	// Celestica Requirement
				dsHmiUserReg.AReActorType[iUM_SelectedLoginNameId]				:= sUM_NewUserActorType;			// Celestica Requirement
				dsHmiUserReg.ARsLastName[iUM_SelectedLoginNameId]				:= sUM_NewUserLastName;
				dsHmiUserReg.ARsFirstName[iUM_SelectedLoginNameId]				:= sUM_NewUserFirstName;
				dsHmiUserReg.ARsLoginName[iUM_SelectedLoginNameId]				:= sUM_NewUserLoginName;			// Same as Username
				//dsHmiUserReg.ARbUserStatus[iUM_SelectedLoginNameId]			:= TRUE;							// 0 = Deactivated/Disable, 1 = Active User
				
				dsHmiUserReg.ARiUserGroupID[iUM_SelectedLoginNameId]			:= sUM_NewUserGroupId;				// Define in HMI TF1800
				dsHmiUserReg.ARwsUserGroupName[iUM_SelectedLoginNameId]			:= ARsUserGroup[sUM_NewUserGroupId];// Define in HMI TF1800
				
				IF sUM_NewPassword <> '' THEN
					dsHmiUserReg.ARsPw[iUM_SelectedLoginNameId]						:= sUM_NewPassword;		// It will only update the password if the New and Confirm password filled accurately.
				END_IF
				
				sMessage := 'User Info is Updated successfully. Please go to Login page to proceed';	
				iUM_SelectedLoginNameId := 0;	
				iCase := 8; // Clear new user registration field and return
	
			END_IF
				
		ELSIF bUM_ReturnPBRE.Q THEN

			sMessage := 'Returned';	
			iUM_SelectedLoginNameId := 0;	
			iCase := 8; // Clear and return

		END_IF		
	51: // User Management -> Delete User 
	
		sMessage := 'Are you sure you want to DELETE selected user?';	
	
		IF bUM_ConfirmPBRE.Q THEN 
					
			dsHmiUserReg.ARsOperatorIdentifier[iUM_SelectedLoginNameId]		:= '';				// Celestica Requirement
			dsHmiUserReg.AReActorType[iUM_SelectedLoginNameId]				:= 0;				// Celestica Requirement
			dsHmiUserReg.ARsLastName[iUM_SelectedLoginNameId]				:= '';
			dsHmiUserReg.ARsFirstName[iUM_SelectedLoginNameId]				:= '';
			dsHmiUserReg.ARsLoginName[iUM_SelectedLoginNameId]				:= '';				// Same as Username
			dsHmiUserReg.ARbUserStatus[iUM_SelectedLoginNameId]				:= FALSE;			// 0 = Deactivated/Disable, 1 = Active User
			
			dsHmiUserReg.ARiUserGroupID[iUM_SelectedLoginNameId]			:= 0;				// Define in HMI TF1800
			dsHmiUserReg.ARwsUserGroupName[iUM_SelectedLoginNameId]			:= TO_WSTRING('');	// Define in HMI TF1800
			dsHmiUserReg.ARsPw[iUM_SelectedLoginNameId]						:= '';					

			sMessage := 'Selected user has been DELETED.';
			iUM_SelectedLoginNameId := 0;	
			iCase := 0;
		
		ELSIF bUM_ReturnPBRE.Q THEN

			sMessage := 'Returned';	
			iUM_SelectedLoginNameId := 0;	
			iCase := 0;

		END_IF

	61: // User Management -> Temporary Disable selected User 
	
		IF bUM_EnablePBRE.Q THEN
			 sMessage := 'Are you sure you want to ENABLE selected user?';	

		ELSIF bUM_DisablePBRE.Q THEN
			 sMessage := 'Are you sure you want to DISABLE selected user?';	
		END_IF
	

	
		IF bUM_ConfirmPBRE.Q AND sMessage = 'Are you sure you want to ENABLE selected user?' THEN 
					
			dsHmiUserReg.ARbUserStatus[iUM_SelectedLoginNameId]				:= TRUE;			// 0 = Deactivated/Disable, 1 = Active User			
			sMessage := 'Selected user has been ENABLE.';	
			iUM_SelectedLoginNameId := 0;	
			iCase := 0;
		
		ELSIF bUM_ConfirmPBRE.Q AND sMessage = 'Are you sure you want to DISABLE selected user?' THEN 			
					
			dsHmiUserReg.ARbUserStatus[iUM_SelectedLoginNameId]				:= FALSE;			// 0 = Deactivated/Disable, 1 = Active User			
			sMessage := 'Selected user has been DISABLE.';	
			iUM_SelectedLoginNameId := 0;	
			iCase := 0;
		
		ELSIF bUM_ReturnPBRE.Q THEN

			sMessage := 'Returned';	
			iUM_SelectedLoginNameId := 0;	
			iCase := 0;

		END_IF

END_CASE



// Clear Message after x period of time
	
	sMessageDelayTimer(IN:=sMessage <> '' AND iCase <> 42 AND iCase <> 51 AND iCase <> 61 , PT:=T#3S , Q=> , ET=> );
	IF sMessageDelayTimer.Q THEN
		sMessage := '';
	END_IF

END_FUNCTION_BLOCK

// ---- FBs/FB_Others TBD/fbV3_XML_Handler.TcPOU
FUNCTION_BLOCK fbV3_XML_Handler
VAR_INPUT

	bEnable							: BOOL; (* Input *)
	bFBInterlock						: BOOL; (* Input *)
	sFileLocation						: STRING := 'C:\JKS\ImportExport_XMLserver\'; (* Input *)
	sFilename						: STRING := 'ProductRecipe'; (* Input *)
	bAddRecipeNoToFilenameEn 		: BOOL; (* Input *)

	bErrorRst						: BOOL; (*Input*)

	iXMLRecipeNo_Input				: INT; (*Input*)
	bCompleteAutoResetEn			: BOOL;
	i_AutoCompleteDelayTime_Sec		: INT := 2;
END_VAR
VAR_IN_OUT
	iImport_ReplaceHS				: INT; (* In_Out *) (*0-Idle, 1-Enable, 2-Busy, 3-Done, 4-Error*)  (*Import or Replaced from XML to Internal Memory with Specified Recipe No*)
	iExportHS						: INT; (* In_Out *) (*0-Idle, 1-Enable, 2-Busy, 3-Done, 4-Error*)  (*Export to XML From Internal Memory with Specified Recipe No*)
	iDeleteAllHS						: INT; (* In_Out *) (*0-Idle, 1-Enable, 2-Busy, 3-Done, 4-Error*)  (*Delete ALL Recipe Internal Memory*)

END_VAR
VAR_OUTPUT
	bBusyFlag						: BOOL; (* Output *) (* Need to place at "bFBInterlock" as "Interlock" if the program applied more than 1 FB*)
	bErrorFlag						: BOOL; (* Output *) (* Error Indication*)
	udErrorID						: UDINT; (*Output *)

END_VAR
VAR

	udImportErrID					: UDINT;
	udExportErrID					: UDINT;

	bImportEn					: BOOL;
	bExportEn					: BOOL;

	bImportBusyFlag				: BOOL;
	bExportBusyFlag				: BOOL;

	bImportCompletedFlag			: BOOL;
	bExportCompletedFlag			: BOOL;

	bImportErrorFlag				: BOOL;
	bExportErrorFlag				: BOOL;

(*	sImportMsg					: STRING;
	sExportMsg					: STRING; *)


	iTask						: INT := 1;
	iCase_Fun					: INT := 1;
	iCase_Import					: INT;
	iCase_Export					: INT;
	iCase_Delete					: INT;
	fbV3ImportExportXML 			: fbV3_ImportExportXML;


	sFbFilePath					:T_MaxString;
	sFbXPath					:T_MaxString(* := '/Recipe/Parameter'*);
	bFbImport					: BOOL;
	bFbExport					: BOOL;
	bFbErrorReset				: BOOL;

	bFbReadDone				: BOOL;
	bFbReadBusy				: BOOL;
	bFbReadError				: BOOL;
	udFbReadErrorID				: UDINT;

	bFbWriteDone				: BOOL;
	bFbWriteBusy				: BOOL;
	bFbWriteError				: BOOL;
	udFbWriteErrorID				: UDINT;

	bFbReadErrorRE				: R_TRIG;
	bFbWriteErrorRE				: R_TRIG;
(*	iFbReadCount				: INT;
	iFbWriteCount				: INT;

	tSecsGemLoadSimulateTimer	: TON;
*)	ARiSubActionEmpty			: ARRAY [1..10] OF INT;

	iImport_ReplaceHSErrorFE			: F_TRIG;
	iExportHSErrorFE					: F_TRIG;
	iDeleteAllHSErrorFE				: F_TRIG;
	iImport_ReplaceHSCompleteRE		: R_TRIG;
	iDeleteAllHSCompleteRE			: R_TRIG;

	sFileLocation_Int: STRING;
	sFilename_Int: STRING;
	tAutoCompleteDelayTimer: TON;
END_VAR


	IF iImport_ReplaceHS <> 0 OR iExportHS <> 0 OR  iDeleteAllHS <> 0 THEN
	bBusyFlag := TRUE;
	ELSE
	bBusyFlag := FALSE;
	END_IF

	IF bBusyFlag THEN
	iXMLRecipeNo := iXMLRecipeNo_Input;
	END_IF

	IF iImport_ReplaceHS = 4 OR iExportHS = 4 OR  iDeleteAllHS = 4 THEN
	bErrorFlag := TRUE;
	ELSE
	bErrorFlag := FALSE;
	END_IF

	IF iImport_ReplaceHS = 4 THEN
	udErrorID := udImportErrID;
	ELSIF iExportHS = 4 THEN
	udErrorID := udExportErrID;
	ELSE
	udErrorID := 0;
	END_IF

	tAutoCompleteDelayTimer(IN:= iImport_ReplaceHS = 3 OR iExportHS = 3 OR  iDeleteAllHS = 3 , PT:= INT_TO_TIME(i_AutoCompleteDelayTime_Sec)*1000 , Q=> , ET=> );

	IF iImport_ReplaceHS = 3 AND tAutoCompleteDelayTimer.Q THEN
		iImport_ReplaceHS 	:= 0;

	ELSIF iExportHS = 3 AND tAutoCompleteDelayTimer.Q THEN
		iExportHS 			:= 0;

	ELSIF iDeleteAllHS = 3 AND tAutoCompleteDelayTimer.Q THEN
		iDeleteAllHS 			:= 0;

	END_IF




	IF bEnable AND NOT bFBInterlock THEN

		Action_Export();
		Action_ImportReplace();
		Action_DeleteAll();
		ImportExportXML();

		IF bErrorRst THEN

			IF iImport_ReplaceHS = 4 THEN
				iImport_ReplaceHS := 0;
			ELSIF iExportHS = 4 THEN
				iExportHS := 0;
			ELSIF iDeleteAllHS = 4 THEN
				iDeleteAllHS := 0;
			END_IF
		END_IF

		iImport_ReplaceHSErrorFE(CLK:= iImport_ReplaceHS = 4  , Q=> );
		iExportHSErrorFE(CLK:= iExportHS = 4  , Q=> );
		iDeleteAllHSErrorFE(CLK:= iDeleteAllHS = 4  , Q=> );

		IF iImport_ReplaceHSErrorFE.Q OR iExportHSErrorFE.Q OR iDeleteAllHSErrorFE.Q OR bErrorRst THEN
		bFbErrorReset := TRUE;
		ELSE
		bFbErrorReset := FALSE;
		END_IF

		iImport_ReplaceHSCompleteRE(CLK:= iImport_ReplaceHS = 3  , Q=> );
		iDeleteAllHSCompleteRE(CLK:= iDeleteAllHS = 3  , Q=> );

		IF iImport_ReplaceHSCompleteRE.Q OR iDeleteAllHSCompleteRE.Q THEN
		bRecipeLoadPB := TRUE;
		END_IF

	END_IF

ACTION Action_DeleteAll:
(*Delete 					- DeleteAllRecipe  -  S7F17 / S7F18	*)
(* iDeleteAllHS	 		: 0-Idle, 1-Enable, 2-Busy, 3-Done, 4-Error *)
(* iSubAction				: 0-Idle, 1-Import, 2-Export, 3-Clear/Delete 8-Done *)

	IF iDeleteAllHS = 0 THEN
		iCase_Delete := 0;
	END_IF

	CASE iCase_Delete OF

	0:
		IF iDeleteAllHS = 1 THEN
			iCase_Delete := 11; (* Delete Actual Memory #1*)
			ARiSubAction[1] := 3;
			iDeleteAllHS := 2; (* Indicate Busy *)
		END_IF

	11: (* Delete Actual Memory #1*)

		IF ARiSubAction[1] = 8 THEN
		iCase_Delete := 12;
		ARiSubAction[1] := 0;
		ARiSubAction[2] := 3;
		END_IF

	12: (* Delete Actual Memory #2*)

		IF ARiSubAction[2] = 8 THEN
		iCase_Delete := 13;
		ARiSubAction[2] := 0;
		ARiSubAction[3] := 3;
		END_IF

	13: (* Delete Actual Memory #3*)

		IF ARiSubAction[3] = 8 THEN
		iCase_Delete := 18;
		iDeleteAllHS := 3; (*Done*)
		END_IF


	18: (* Completed *)

		ARiSubAction := ARiSubActionEmpty;

	END_CASE
END_ACTION

ACTION Action_Export:
(*Export			 		- Export  -   From IPC to Server - S7F5 / S7F6 *)
(* iExportHS			 	: 0-Idle, 1-Enable, 2-Busy, 3-Done, 4-Error *)
(* iSubAction				: 0-Idle, 1-Import, 2-Export, 3-Clear/Delete 8-Done *)


	IF iExportHS = 0 THEN
		iCase_Export := 0;
	END_IF

	CASE iCase_Export OF

	0:
		IF iExportHS = 1 THEN
			iCase_Export := 11; (* Transfer from Buffer to Actual Memory #1*)
			ARiSubAction[1] := 2;
			iExportHS := 2; (* Indicate Busy *)
		END_IF

	11: (* Transfer from Actual Memory to Buffer #1*)

		IF ARiSubAction[1] = 8 THEN
		iCase_Export := 12;
		ARiSubAction[1] := 0;
		ARiSubAction[2] := 2;
		END_IF

	12: (* Transfer from Actual Memory to Buffer #2*)

		IF ARiSubAction[2] = 8 THEN
		iCase_Export := 13;
		ARiSubAction[2] := 0;
		ARiSubAction[3] := 2;
		END_IF

	13: (* Transfer from Actual Memory to Buffer #3*)

		IF ARiSubAction[3] = 8 THEN
		iCase_Export := 14;
		ARiSubAction[3] := 0;
		END_IF

	14: (* Start Export from Buffer Memory to File*)

		bExportEn := TRUE;

		IF bExportCompletedFlag THEN
		bExportEn := FALSE;
		iCase_Export := 18;
		iExportHS := 3; (*Done*)

		ELSIF bExportErrorFlag THEN
		bExportEn := FALSE;
		iCase_Export := 19; (*Error*)
		iExportHS := 4; (*Error*)
		END_IF



	18: (* Completed *)

		ARiSubAction := ARiSubActionEmpty;

	19: (* Error *)

		ARiSubAction := ARiSubActionEmpty;

	END_CASE
END_ACTION

ACTION Action_ImportReplace:
(*iImport_Replace			 - Import  	-   From Server to IPC - S7F3 / S7F4 *)
(* iImport_ReplaceHS	 	: 0-Idle, 1-Enable, 2-Busy, 3-Done, 4-Error *)
(* iSubAction				: 0-Idle, 1-Import, 2-Export, 3-Clear/Delete 8-Done *)

	IF iImport_ReplaceHS = 0 THEN
		iCase_Import := 0;
	END_IF

	CASE iCase_Import OF

	0:
		IF iImport_ReplaceHS = 1 THEN
			iCase_Import := 11; (* Start Import from File to Buffer Memory*)
			iImport_ReplaceHS := 2; (* Indicate Busy *)
		END_IF

	11: (* Start Import from File to Buffer Memory*)

		bImportEn := TRUE;

		IF bImportCompletedFlag THEN
		bImportEn := FALSE;
		iCase_Import := 12;
		ARiSubAction[1] := 1;

		ELSIF bImportErrorFlag THEN
		bImportEn := FALSE;
		iCase_Import := 19; (*Error*)
		iImport_ReplaceHS := 4; (*Error*)

		END_IF

	12: (* Transfer from Buffer to Actual Memory #1*)

		IF ARiSubAction[1] = 8 THEN
		iCase_Import := 13;
		ARiSubAction[1] := 0;
		ARiSubAction[2] := 1;
		END_IF

	13: (* Transfer from Buffer to Actual Memory #2*)

		IF ARiSubAction[2] = 8 THEN
		iCase_Import := 14;
		ARiSubAction[2] := 0;
		ARiSubAction[3] := 1;
		END_IF

	14: (* Transfer from Buffer to Actual Memory #3*)

		IF ARiSubAction[3] = 8 THEN
		iCase_Import := 18;
		ARiSubAction[3] := 0;
		iImport_ReplaceHS := 3; (*Done*)
		END_IF

	18: (* Completed *)

		ARiSubAction := ARiSubActionEmpty;


	19: (* Error *)

		ARiSubAction := ARiSubActionEmpty;

	END_CASE
END_ACTION

ACTION ImportExportXML:
(* Function Export/Import Between XML to Buffer Memory *)


	fbV3ImportExportXML(
		sFbFilePath		:= sFbFilePath,
		sFbXPath		:= sFbXPath,
		bFbImport		:= bFbImport,
		bFbExport		:= bFbExport,
		bFbErrorReset	:= bFbErrorReset,

		bFbReadDone	=> bFbReadDone,
		bFbReadBusy	=> bFbReadBusy,
		bFbReadError	=> bFbReadError,
		udFbReadErrorID	=> udFbReadErrorID,

		bFbWriteDone	=> bFbWriteDone,
		bFbWriteBusy	=> bFbWriteBusy,
		bFbWriteError	=> bFbWriteError,
		udFbWriteErrorID	=> udFbWriteErrorID);


(*** ImportEn & OutputEn Control ***)

		IF NOT bImportEn AND NOT bExportEn AND NOT bImportErrorFlag AND NOT bExportErrorFlag THEN
		iCase_Fun := 0;
		END_IF



		CASE iCase_Fun OF
		
		0:(* Idling *)
				bFbImport := FALSE;
				bFbExport := FALSE;
				iTask := 0;
				bImportBusyFlag				:= FALSE;
				bExportBusyFlag				:= FALSE;

				bImportCompletedFlag			:= FALSE;
				bExportCompletedFlag			:= FALSE;

				bImportErrorFlag				:= FALSE;
				bExportErrorFlag				:= FALSE;

				udImportErrID					:= 0;
				udExportErrID					:= 0;

				IF bImportEn OR bExportEn THEN
					iTask := 1;
					iCase_Fun := 1;
				END_IF

		1: (* Import/Export Preparation*)
				IF iTask = 1 THEN
				FBXmlSrvRead.pSymAddr:= ADR(DSV3XML_Recipe);
				FBXmlSrvRead.cbSymSize:=SIZEOF(DSV3XML_Recipe);
				FBXmlSrvWrite.pSymAddr:= ADR(DSV3XML_Recipe);
				FBXmlSrvWrite.cbSymSize:=SIZEOF(DSV3XML_Recipe);

				sFileLocation_int := sFileLocation;

				IF bAddRecipeNoToFilenameEn THEN
				sFilename_int := CONCAT(CONCAT(CONCAT(CONCAT(sFilename,'['), INT_TO_STRING(iXMLRecipeNo_Input)),']'),'.xml');
				ELSE
				sFilename_int := CONCAT(sFilename,'.xml');
				END_IF

				sFbXPath := '/ProductRecipe/Parameter';

				END_IF

				sFbFilePath := CONCAT(sFileLocation_Int,sFilename_Int);
		
				IF iTask <= 1 THEN
					IF bImportEn THEN
						iCase_Fun := 11;
						bImportBusyFlag := TRUE;
					ELSIF bExportEn THEN
						iCase_Fun := 21;
						bExportBusyFlag := TRUE;
					END_IF
				ELSE
				iCase_Fun := 30; (*Trigger Completion*)
				END_IF
		
		11: (* Import Step 1 *)
				bFbImport := TRUE;
		
				IF NOT bFbReadBusy AND bFbReadDone THEN
				iCase_Fun := 12;
				ELSIF bFbReadError THEN
				iCase_Fun := 19;
				END_IF
		
		12: (* Import Step 2 *)

				bFbImport := FALSE;
		
				IF NOT bFbReadDone THEN

						iTask := iTask + 1;
						iCase_Fun := 1;

				END_IF

		
		
		21: (* Export Step 1 *)
				bFbExport := TRUE;

				IF NOT bFbWriteBusy AND bFbWriteDone THEN
				iCase_Fun := 22;
				ELSIF bFbWriteError THEN
				iCase_Fun := 29;
				END_IF
		
		22: (* Export Step 2 *)
				bFbExport := FALSE;

				IF NOT bFbWriteDone THEN

						iTask := iTask + 1;
						iCase_Fun := 1;

				END_IF
		
		

		19:; (* Read Error *)
				bImportErrorFlag 				:= bFbReadError;
				udImportErrID 				:= udFbReadErrorID;
				bImportBusyFlag				:= FALSE;
				bFbImport 					:= FALSE;


		29:; (* Write Error *)
				bExportErrorFlag 				:= bFbWriteError;
				udExportErrID 				:= udFbWriteErrorID;
				bExportBusyFlag				:= FALSE;
				bFbExport 					:= FALSE;

		
		30:; (* Import/Export Completed - DONE *)
				IF bImportEn THEN bImportCompletedFlag := TRUE; bImportBusyFlag := FALSE;
				ELSIF bExportEn THEN bExportCompletedFlag := TRUE; bExportBusyFlag := FALSE;
				END_IF

		END_CASE
END_ACTION

END_FUNCTION_BLOCK

// ---- FBs/FB_Others TBD/fbV3_ImportExportXML.TcPOU
FUNCTION_BLOCK fbV3_ImportExportXML
VAR_INPUT
	sFbFilePath					:T_MaxString;
	sFbXPath					:T_MaxString; (* Default ->    '/L1/L2/L3/L4/L5/L6/L7/L8/L9'  *)
	bFbImport					: BOOL;
	bFbExport					: BOOL;
	bFbErrorReset				: BOOL;

END_VAR

VAR_OUTPUT
	bFbReadDone				: BOOL;
	bFbReadBusy				: BOOL;
	bFbReadError				: BOOL;
	udFbReadErrorID				: UDINT;

	bFbWriteDone				: BOOL;
	bFbWriteBusy				: BOOL;
	bFbWriteError				: BOOL;
	udFbWriteErrorID				: UDINT;
END_VAR

VAR
	bFbEXERead				: BOOL;
	bFbEXEWrite					: BOOL;

	eFbPath 						: E_OpenPath := PATH_GENERIC;

	step							: INT;
	bFbErrorResetRE				: R_TRIG;
END_VAR

bFbErrorResetRE(CLK:=bFbErrorReset , Q=> );


CASE step OF


0:	(*Initialize*)

	FBXmlSrvRead.bExecute		:=FALSE;
	FBXmlSrvWrite.bExecute		:=FALSE;
	bFbEXERead				:=FALSE;
	bFbEXEWrite					:=FALSE;

	bFbReadBusy				:= FALSE;
	bFbReadError				:= FALSE;
	udFbReadErrorID				:= 0;

	bFbWriteBusy				:= FALSE;
	bFbWriteError				:= FALSE;
	udFbWriteErrorID				:= 0;


	IF bFbImport THEN
	bFbReadDone 				:=FALSE;
	bFbEXERead				:=TRUE;
	step							:=1;
	END_IF

	IF bFbExport THEN
	bFbWriteDone				:=FALSE;
	bFbEXEWrite					:= TRUE;
	step							:=2;
	END_IF

1:	(* Read XML function block*)


		IF NOT bFbEXERead THEN

			IF NOT FBXmlSrvRead.bBusy AND NOT FBXmlSrvRead.bError THEN
			step:=10;
			END_IF

			IF bFbErrorResetRE.Q AND FBXmlSrvRead.bError THEN
			step:=0;
			END_IF

		END_IF

		FBXmlSrvRead(
		ePath		:=eFbPath ,
		nMode		:=XMLSRV_ADDMISSING ,
	(*	pSymAddr	:= ADR(StDataTransfer),
		cbSymSize	:=SIZEOF(StDataTransfer) ,*)
		sFilePath	:=sFbFilePath ,
		sXPath		:=sFbXPath ,
		bExecute	:= bFbEXERead,
		bBusy		 => bFbReadBusy,
		bError 		=> bFbReadError,
		nErrId 		=> udFbReadErrorID);

		bFbEXERead := FALSE;


10: (*Mapping*)

		bFbReadDone	:=TRUE;

		IF NOT bFbImport THEN
		bFbReadDone:=FALSE;
		step:=0;
		END_IF

2: (* Write XML function block*)

		IF NOT bFbEXEWrite THEN

			IF NOT FBXmlSrvWrite.bBusy AND NOT FBXmlSrvWrite.bError THEN
			step:=20;
			END_IF

			IF bFbErrorResetRE.Q AND FBXmlSrvWrite.bError THEN
			step:=0;
			END_IF

		END_IF

		FBXmlSrvWrite(
		ePath:=eFbPath ,
		nMode:=XMLSRV_ADDMISSING ,
(*		pSymAddr:=ADR(XML_ImportExport) ,
		cbSymSize:=SIZEOF(XML_ImportExport) ,*)
		sFilePath:=sFbFilePath ,
		sXPath:= sFbXPath,
		bExecute:=bFbEXEWrite,
		bBusy => bFbWriteBusy,
		bError => bFbWriteError,
		nErrId => udFbWriteErrorID);

		bFbEXEWrite := FALSE;



20:  (* Mapping*)

		bFbWriteDone:=TRUE;

		IF NOT bFbExport THEN
		bFbWriteDone:=FALSE;
		step:=0;
		END_IF

END_CASE

END_FUNCTION_BLOCK

// ---- FBs/B_JKS_CustomFB/fbArmCtrlFolder/AM_MoveAbsolute.TcPOU
FUNCTION_BLOCK AM_MoveAbsolute
VAR_INPUT
	bEnable	: BOOL;
	iDistance	: INT;
	i1stRPM		: INT;
	i2ndRPM		: INT;
	i2ndSpdRange	: INT;
	iOffSetRange		: INT;
	iRatio			: REAL;
	iDtime			: INT;
	iDStep			: INT;
	MasterActualPosition	: LREAL;

END_VAR
VAR_OUTPUT
	bDone			: BOOL;
	bMoveFor		: BOOL;
	bMoveRev		: BOOL;
	iSpeedOut		: INT;



END_VAR
VAR
	RAP1: MC_ReadActualPosition;
	SpdRangeN: INT;
	SpdRangeP: INT;
	SpeedEnable: BOOL;
	OffSetN: INT;
	OffSetP: INT;
	OffSetEnable: BOOL;
	DisEn: BOOL;
	RPM1En: BOOL;
	RPM2En: BOOL;
	PosCmp1: fbServoPosCmp;
	ArmInRange: BOOL;
	RpmConvert: AM_InverterConversionHz;
	RpmConvert1: AM_InverterConversionHz;
	PosCmp2: fbServoPosCmp;
	TriggerMovFor: BOOL;
	TriggerStandStill: BOOL;
	TriggerMovRev: BOOL;
	TRIG1: R_TRIG;
	MoveEnable: BOOL;
	i1stSpeedOut : INT;
	i2ndSpeedOut : INT;
	bMoveForInt: BOOL;
	bMoveRevInt: BOOL;
	MotorMovingProfileFB: fbIndMotDecCtrl;
	PerSpd: INT;
END_VAR
VAR // added by the converter: edge detectors and wires of the graphical bodies
    _w1 : BOOL;
    _w2, _w3 : INT;
END_VAR

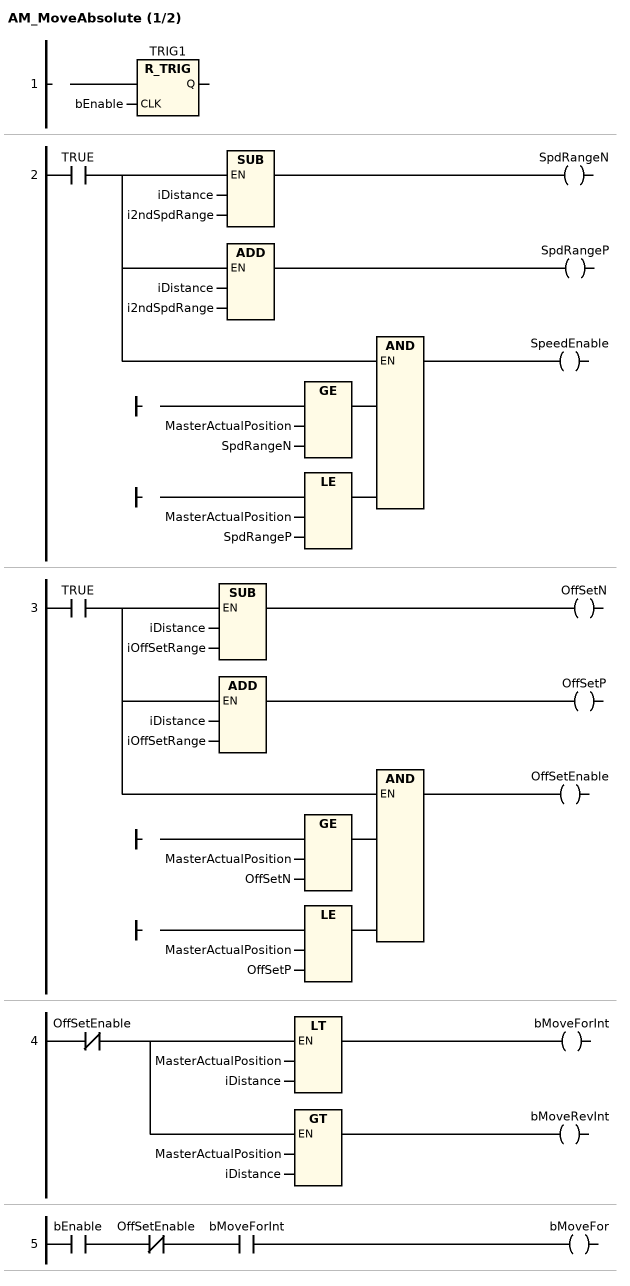
// NETWORK 1
TRIG1(CLK := bEnable); // R_TRIG

// NETWORK 2
SpdRangeN := iDistance - i2ndSpdRange;
SpdRangeP := iDistance + i2ndSpdRange;
SpeedEnable := MasterActualPosition >= SpdRangeN AND MasterActualPosition <= SpdRangeP;

// NETWORK 3
OffSetN := iDistance - iOffSetRange;
OffSetP := iDistance + iOffSetRange;
OffSetEnable := MasterActualPosition >= OffSetN AND MasterActualPosition <= OffSetP;

// NETWORK 4
_w1 := NOT OffSetEnable;
bMoveForInt := _w1 AND MasterActualPosition < iDistance;
bMoveRevInt := _w1 AND MasterActualPosition > iDistance;

// NETWORK 5
bMoveFor := bEnable AND NOT OffSetEnable AND bMoveForInt;

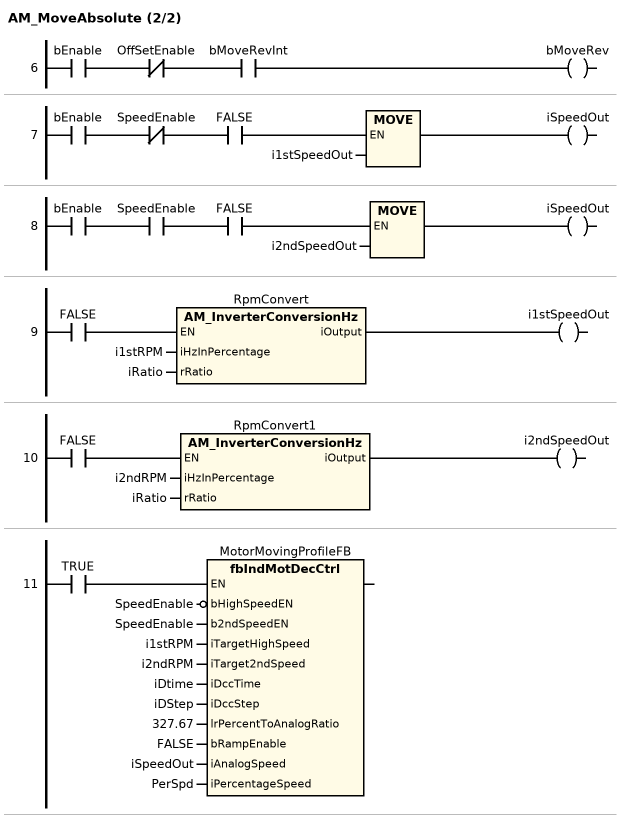
// NETWORK 6
bMoveRev := bEnable AND NOT OffSetEnable AND bMoveRevInt;

// NETWORK 7
IF bEnable AND NOT SpeedEnable AND FALSE THEN _w2 := i1stSpeedOut; END_IF
iSpeedOut := _w2;

// NETWORK 8
IF bEnable AND SpeedEnable AND FALSE THEN _w3 := i2ndSpeedOut; END_IF
iSpeedOut := _w3;

// NETWORK 9
IF FALSE THEN
    RpmConvert(iHzInPercentage := i1stRPM, rRatio := iRatio); // AM_InverterConversionHz
END_IF
i1stSpeedOut := RpmConvert.iOutput;

// NETWORK 10
IF FALSE THEN
    RpmConvert1(iHzInPercentage := i2ndRPM, rRatio := iRatio); // AM_InverterConversionHz
END_IF
i2ndSpeedOut := RpmConvert1.iOutput;

// NETWORK 11
MotorMovingProfileFB(
    bHighSpeedEN := NOT SpeedEnable,
    b2ndSpeedEN := SpeedEnable,
    iTargetHighSpeed := i1stRPM,
    iTarget2ndSpeed := i2ndRPM,
    iDccTime := iDtime,
    iDccStep := iDStep,
    lrPercentToAnalogRatio := 327.67,
    bRampEnable := FALSE,
    iAnalogSpeed := iSpeedOut,
    iPercentageSpeed := PerSpd); // fbIndMotDecCtrl

END_FUNCTION_BLOCK

// ---- FBs/B_JKS_CustomFB/fbArmCtrlFolder/fbServoPosCmp.TcPOU
FUNCTION_BLOCK fbServoPosCmp
VAR_INPUT

	Enable : BOOL;
	Data1_Lreal : LREAL;
	Data1Range : LREAL;
	ActualData : LREAL;


END_VAR
VAR_OUTPUT

	bInRange : BOOL;

END_VAR
VAR
	Data1Low: LREAL;
	Data1High: LREAL;
	LowInRange: BOOL;
	HighInRange: BOOL;
END_VAR

Data1Low := (Data1_Lreal - Data1Range);
Data1High := (Data1_Lreal + Data1Range);

IF ActualData > Data1Low THEN
LowInRange := TRUE;
ELSE
LowinRange := FALSE;
END_IF

IF ActualData < Data1High THEN
HighInRange := TRUE;
ELSE
HighInRange := FALSE;
END_IF

IF Enable AND LowInRange AND HighInRange THEN
bInRange := TRUE;
ELSE
bInRange := FALSE;
END_IF

END_FUNCTION_BLOCK

// ---- FBs/B_JKS_CustomFB/fbConversionCtrl/AM_InverterConversionHz.TcPOU
FUNCTION_BLOCK AM_InverterConversionHz
VAR_INPUT
	iHzInPercentage		: INT;
	rRatio				: REAL;
END_VAR
VAR_OUTPUT
	iOutput				: INT;
END_VAR
VAR
	rHzInPercentage: REAL;
	rResult: REAL;
END_VAR

rHzInPercentage := INT_TO_REAL(iHzInPercentage);

rResult := (rHzInPercentage*rRatio);

iOutput := REAL_TO_INT(rResult);

END_FUNCTION_BLOCK

// ---- FBs/B_JKS_CustomFB/fbArmCtrlFolder/fbIndMotDecCtrl.TcPOU
FUNCTION_BLOCK fbIndMotDecCtrl
VAR_INPUT
	bHighSpeedEN : BOOL;
	b2ndSpeedEN : BOOL;
	iTargetHighSpeed : INT;
	iTarget2ndSpeed : INT;
	iDccTime : INT;
	iDccStep : INT;
	lrPercentToAnalogRatio : LREAL;
	bRampEnable : BOOL;

END_VAR
VAR_OUTPUT


END_VAR

VAR_IN_OUT
	iAnalogSpeed : INT;
	iPercentageSpeed : INT;
END_VAR

VAR
	tRefreshTime: TIME;
	RefreshTimer: TON;
	RefreshTimerRE: R_TRIG;
	lrAnalogSpeed : LREAL;


	iValueToDeduce: INT;
	iPercentPerStep: INT;
	iRampValue: INT;
	b2ndSpeedRE: R_TRIG;
END_VAR

(*  No EN Signal for both HighSpeed and 2ndSpeed *)
IF NOT  bHighSpeedEN AND NOT b2ndSpeedEN THEN
iPercentageSpeed := 0;
END_IF

(* HighSpeed Enable *)
IF bHighSpeedEN AND NOT b2ndSpeedEN THEN
iPercentageSpeed := iTargetHighSpeed;
END_IF

(*Convertion from Percentage to Analog *)
IF lrPercentToAnalogRatio > 0 AND iPercentageSpeed > 0 THEN
lrAnalogSpeed := lrPercentToAnalogRatio * INT_TO_LREAL(iPercentageSpeed);
ELSE
lrAnalogSpeed := 0;
END_IF

iAnalogSpeed := LREAL_TO_INT(lrAnalogSpeed);


(* 2ndSpeed Enable *)
IF NOT b2ndSpeedEN THEN
iRampValue := 0;
END_IF

IF iTargetHighSpeed > 0 AND iTarget2ndSpeed > 0 AND iDccStep > 0 THEN
iPercentPerStep := (iTargetHighSpeed - iTarget2ndSpeed)/iDccStep;
END_IF

IF iDccTime > 0 AND iDccStep > 0 THEN
tRefreshTime := INT_TO_TIME(iDccTime*1000/iDccStep);
END_IF

IF b2ndSpeedEN AND NOT bHighSpeedEN AND bRampEnable THEN

	IF iPercentageSpeed > iTarget2ndSpeed THEN
		RefreshTimer(IN:=NOT RefreshTimer.Q , PT:= tRefreshTime , Q=> , ET=> );
		RefreshTimerRE(CLK:=RefreshTimer.Q , Q=> );
	END_IF

b2ndSpeedRE(CLK:=b2ndSpeedEN , Q=> );

	IF b2ndSpeedRE.Q THEN
	iRampValue := 0;
	END_IF

	IF RefreshTimerRE.Q AND iPercentageSpeed > iTarget2ndSpeed THEN
	iRampValue := iRampValue + iPercentPerStep;
	END_IF

iPercentageSpeed := iTargetHighSpeed - iRampValue;

END_IF

IF NOT bRampEnable THEN
	IF b2ndSpeedEN THEN
	iPercentageSpeed := iTarget2ndSpeed;
	END_IF
END_IF

END_FUNCTION_BLOCK

// ---- FBs/B_JKS_CustomFB/fbArmCtrlFolder/fbArmMoveInterLock.TcPOU
FUNCTION_BLOCK fbArmMoveInterLock
VAR_INPUT
	diArmPosVariable		: DINT;


END_VAR
VAR_IN_OUT

	diArmInterlock	: DINT;

END_VAR
VAR

	InterlockEn: BOOL;
END_VAR
VAR // added by the converter: edge detectors and wires of the graphical bodies
    _w1 : ANY;
END_VAR

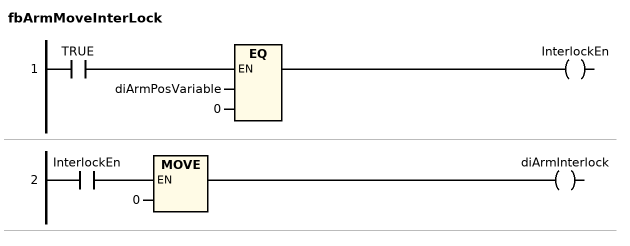
// NETWORK 1
InterlockEn := diArmPosVariable = 0;

// NETWORK 2
IF InterlockEn THEN _w1 := 0; END_IF
diArmInterlock := _w1;

END_FUNCTION_BLOCK

// ---- FBs/B_JKS_CustomFB/fbArmCtrlFolder/fbArmPnpCtrl.TcPOU
FUNCTION_BLOCK fbArmPnpCtrl
VAR_INPUT
	bEN									:	BOOL;
(*	bExternalCtrl							: 	BOOL;
	bPnPStart							:	BOOL;
	iPickStnNo							:	INT;
	iTransferStnNo						:	INT;
*)	bReset								:	BOOL;
	bMovingHalt							:	BOOL;
	iArmNo								:	INT;
	iCurrentHorzZoneNo					:	INT;
	bDownPickCondition					:	BOOL;
	bDownTransferCondition				:	BOOL;
	ARbPickMidDownStnEn				:	ARRAY [0..iStnQty] OF BOOL;
	ARbTransferMidDownStnEn			:	ARRAY [0..iStnQty] OF BOOL;
	ARiStationDippingTime				:	ARRAY [0..iStnQty] OF INT;
	AR3sbArmPositionCFM				:	ARRAY [0..iArmQty,0..iArmStnQty,0..6] OF BOOL; (*1 = UNHOOK,2 = DOWN,3 = HOOK, 4= TOP*)
	iStepDelayTime						:	INT;
END_VAR
VAR_OUTPUT
	bPnpCompleted						:	BOOL;
	bPnPbusy								:	BOOL;
	bArmReady							:  BOOL;
	bMoveTop								:	BOOL;
	bMoveLdDown						:	BOOL;
	bMoveUldDown						:	BOOL;
	ARbMoveStnMidDown				:	ARRAY [0..iStnQty] OF BOOL;
	ARbMoveStnDown					:	ARRAY [0..iStnQty] OF BOOL;
	bMoveLdHook							:	BOOL;
	bMoveUldHook						:	BOOL;
	ARbMoveStnHook						:	ARRAY [0..iStnQty] OF BOOL;
	bMoveLdUnhook						:	BOOL;
	bMoveUldUnhook						:	BOOL;
	ARbMoveStnUnhook					:	ARRAY [0..iStnQty] OF BOOL;
	iPnpStep								: INT;
	tStepDelayTimeEV					: TIME;
	tStationDrippingTimeEV				: TIME;
	sStatusMessage						: STRING(50);

END_VAR

VAR_IN_OUT PERSISTENT
	DSArmBasketInfo	 						: DS_BasketInfo;
	ARiStnNoToCalledArm_Uni					: ARRAY [0..iArmQty] OF INT; 									(*Universal*) (* Output - Link with fbArmPnP, Array based on Arm No, The Int will store which Station that calling the Arm*)
	ARDSGnrFeedArmPnpParameter_Uni		: ARRAY [0..iArmQty] OF DSGnr_CalledArmPnpParameter; 	(*Universal*) (* Output - Link with fbArmPnP, Array based on Current Station No, Arm should move based on this DataStructure Info*)

END_VAR

VAR
	DSEmptyGnrCalledArmPnpParameter : DSGnr_CalledArmPnpParameter;
	bPnpStart_Read_RE: R_TRIG;
	bPnpStart_Read_FE: F_TRIG;
	iResetFL: INT;
	tStepDelay: TON;
	bStepDelayEn: BOOL;
	iPickStnNoInt: INT;
	iTransferStnNoInt: INT;
	iCurrentHorzZoneNoint: INT;
	bDownPickConditionHR: BOOL;
	bDownTransferConditionHR: BOOL;
	bStationDrippingTimeST: BOOL;
	tStationDrippingTime: TON;
	iStationDrippingTimeInt: INT;
	bPnpStart_Read : BOOL;
	iPickStnNo_Read: INT;
	iPickStnNo_ReadInt: INT;
	iTransferStnNo_Read: INT;
	iTransferStnNo_ReadInt: INT;
	iPnpStep5RE: R_TRIG;
END_VAR

(*Mapping*)

iPickStnNo_Read 			:= ARDSGnrFeedArmPnpParameter_Uni[iArmNo].iPickStationNo;
iTransferStnNo_Read 		:= ARDSGnrFeedArmPnpParameter_Uni[iArmNo].iTransferStationNo;

IF ARiStnNoToCalledArm_Uni[iArmNo] <> 0 THEN
bPnpStart_Read := TRUE;
ELSE
bPnpStart_Read := FALSE;
END_IF





(*R_TRIG*)
bPnpStart_Read_RE(CLK:=bPnpStart_Read , Q=> );

(*F_TRIG*)
bPnpStart_Read_FE(CLK:=bPnpStart_Read , Q=> );

(******Station No Conversion******)
(*Pick StnNoConversion*)

IF iPickStnNo_Read = iLdStnID THEN
iPickStnNo_ReadInt := 1;
ELSIF
iPickStnNo_Read = iUldStnID THEN
iPickStnNo_ReadInt := iStnQty+2;
ELSIF
iPickStnNo_Read >= 1 AND iPickStnNo_Read <= iStnQty THEN
iPickStnNo_ReadInt := iPickStnNo_Read+1;
ELSE
iPickStnNo_ReadInt := 0;
END_IF

(*Transfer StnNoConversion*)

IF iTransferStnNo_Read = iLdStnID THEN
iTransferStnNo_ReadInt := 1;
ELSIF
iTransferStnNo_Read = iUldStnID THEN
iTransferStnNo_ReadInt := iStnQty+2;
ELSIF
iTransferStnNo_Read >= 1 AND iTransferStnNo_Read <= iStnQty THEN
iTransferStnNo_ReadInt := iTransferStnNo_Read+1;
ELSE
iTransferStnNo_ReadInt := 0;
END_IF


(*iCurrentHorzZoneNo StnNoConversion*)

IF iCurrentHorzZoneNo = iLdStnID THEN
iCurrentHorzZoneNoint := 1;
ELSIF
iCurrentHorzZoneNo = iUldStnID THEN
iCurrentHorzZoneNoint := iStnQty+2;
ELSIF
iCurrentHorzZoneNo >= 1 AND iCurrentHorzZoneNo <= iStnQty THEN
iCurrentHorzZoneNoint := iCurrentHorzZoneNo+1;
ELSE
iCurrentHorzZoneNoint := 0;
END_IF




(******Sequence Start******)
(*PnpStep Rising Edge*)
iPnpStep5RE(CLK:=iPnpStep = 5 , Q=> );
(*Step Delay Timer*)
tStepDelay(IN:=bEN AND bPnpStart_Read AND bStepDelayEn , PT:=INT_TO_TIME(iStepDelayTime*1000) , Q=> , ET=>tStepDelayTimeEV );

(*Station Dripping Timer*)
IF iPickStnNo_Read >= 1 AND iPickStnNo_Read <= iStnQty THEN
iStationDrippingTimeInt := ARiStationDippingTime[iPickStnNo_Read];
ELSE
iStationDrippingTimeInt := 0;
END_IF

tStationDrippingTime(IN:=bEN AND bPnpStart_Read AND bStationDrippingTimeST , PT:=INT_TO_TIME(iStationDrippingTimeInt*1000) , Q=> , ET=>tStationDrippingTimeEV );


(*Waiting Start Signal and Condition*)
IF bEN THEN

		IF bPnpStart_Read_RE.Q AND iPickStnNo_Read > 0 AND iTransferStnNo_Read > 0 THEN
		iPnpStep := 1;
		bPnPbusy := TRUE;
		END_IF


		CASE iPnpStep OF
		
		10: (*Completed*)
		bPnpCompleted:= TRUE;
		bPnPbusy := FALSE;


		9: (*Move Vertical Top Pos*)
		
			IF NOT AR3sbArmPositionCFM[iArmNo,iTransferStnNo_ReadInt,4] THEN
			bMoveTop := TRUE;
			ELSE
			bMoveTop := FALSE;
			bStepDelayEn := TRUE;
			END_IF
		
			IF AR3sbArmPositionCFM[iArmNo,iTransferStnNo_ReadInt,4] AND tStepDelay.Q AND NOT bMovingHalt THEN
			bStepDelayEn := FALSE;
			iPnpStep := 10;
			END_IF
		
		
		8: (*At Transfer Station - Unhook*)
		
			IF NOT AR3sbArmPositionCFM[iArmNo,iTransferStnNo_ReadInt,1] THEN
		
				IF iTransferStnNo_Read = iLdStnID THEN
				bMoveLdUnhook := TRUE;
				END_IF
		
				IF iTransferStnNo_Read = iUldStnID THEN
				bMoveUldUnhook := TRUE;
				END_IF
		
				IF iTransferStnNo_Read >= 1 AND  iTransferStnNo_Read <= iStnQty THEN
				ARbMoveStnUnhook[iTransferStnNo_Read] := TRUE;
				END_IF
		
			ELSE
		
				IF iTransferStnNo_Read >= 1 AND  iTransferStnNo_Read <= iStnQty THEN
				ARbMoveStnUnhook[iTransferStnNo_Read] := FALSE;
				ELSIF iTransferStnNo_Read = iLdStnID THEN
				bMoveLdUnhook := FALSE;
				ELSIF iTransferStnNo_Read = iUldStnID THEN
				bMoveUldUnhook := FALSE;
				END_IF
		
				bStepDelayEn := TRUE;
		
			END_IF
		
			IF AR3sbArmPositionCFM[iArmNo,iTransferStnNo_ReadInt,1] AND tStepDelay.Q AND NOT bMovingHalt THEN
			bStepDelayEn := FALSE;
			iPnpStep := 9;
			END_IF
		
		
		7: (*Move Vertical Down Pos*)

		IF bDownTransferCondition THEN
		bDownTransferConditionHR := TRUE;
		END_IF

			IF bDownTransferConditionHR AND NOT ARbTransferMidDownStnEn[iTransferStnNo_Read] AND NOT AR3sbArmPositionCFM[iArmNo,iTransferStnNo_ReadInt,2] THEN

				IF iTransferStnNo_Read = iLdStnID THEN
				bMoveLdDown := TRUE;
				END_IF
		
				IF iTransferStnNo_Read = iUldStnID THEN
				bMoveUldDown := TRUE;
				END_IF
		
				IF iTransferStnNo_Read >= 1 AND  iTransferStnNo_Read <= iStnQty  THEN
				ARbMoveStnDown[iTransferStnNo_Read] := TRUE;
				END_IF

			ELSIF bDownTransferConditionHR AND ARbTransferMidDownStnEn[iTransferStnNo_Read] AND NOT AR3sbArmPositionCFM[iArmNo,iTransferStnNo_ReadInt,5] THEN

				IF iTransferStnNo_Read >= 1 AND  iTransferStnNo_Read <= iStnQty  THEN
				ARbMoveStnMidDown[iTransferStnNo_Read] := TRUE;
				END_IF

			END_IF

			IF
			(*bDownTransferConditionHR AND*) NOT ARbTransferMidDownStnEn[iTransferStnNo_Read] AND AR3sbArmPositionCFM[iArmNo,iTransferStnNo_ReadInt,2]
			OR
			(*bDownTransferConditionHR AND*) ARbTransferMidDownStnEn[iTransferStnNo_Read] AND AR3sbArmPositionCFM[iArmNo,iTransferStnNo_ReadInt,5]
			THEN
				IF iTransferStnNo_Read >= 1 AND  iTransferStnNo_Read <= iStnQty THEN
				ARbMoveStnMidDown[iTransferStnNo_Read] := FALSE;
				ARbMoveStnDown[iTransferStnNo_Read] := FALSE;
				ELSIF iTransferStnNo_Read = iLdStnID THEN
				bMoveLdDown := FALSE;
				ELSIF iTransferStnNo_Read = iUldStnID THEN
				bMoveUldDown := FALSE;
				END_IF

				bStepDelayEn := TRUE;

				IF tStepDelay.Q AND NOT bMovingHalt THEN
				bStepDelayEn := FALSE;
				bDownTransferConditionHR := FALSE;
				iPnpStep := 8;
				END_IF

			END_IF

		6: (*Move to Transfer Station - Horizontal Hook Movement*)
		
			IF NOT AR3sbArmPositionCFM[iArmNo,iTransferStnNo_ReadInt,3] THEN
		
				IF iTransferStnNo_Read = iLdStnID THEN
				bMoveLdHook := TRUE;
				END_IF

				IF iTransferStnNo_Read = iUldStnID THEN
				bMoveUldHook := TRUE;
				END_IF
		
				IF iTransferStnNo_Read >= 1 AND  iTransferStnNo_Read <= iStnQty THEN
				ARbMoveStnHook[iTransferStnNo_Read] := TRUE;
				END_IF

			ELSE
		
				IF iTransferStnNo_Read >= 1 AND  iTransferStnNo_Read <= iStnQty THEN
				ARbMoveStnHook[iTransferStnNo_Read] := FALSE;
				ELSIF iTransferStnNo_Read = iLdStnID THEN
				bMoveLdHook := FALSE;
				ELSIF iTransferStnNo_Read = iUldStnID THEN
				bMoveUldHook := FALSE;
				END_IF
		
				bStepDelayEn := TRUE;
		
			END_IF
		
			IF AR3sbArmPositionCFM[iArmNo,iTransferStnNo_ReadInt,3] AND tStepDelay.Q AND NOT bMovingHalt THEN
			bStepDelayEn := FALSE;
			iPnpStep := 7;
			END_IF

		
		5: (*Move Vertical Top Pos*)
		
			(*Addtional Task - Push Station Sequence Recipe No from GnrPnpParameter to Basket Info*)
			DSArmBasketInfo.iStationSeqenceRecipeNo := ARDSGnrFeedArmPnpParameter_Uni[iArmNo].iStnSeqRecipeNo;
			IF iPnpStep5RE.Q THEN
			DSArmBasketInfo.iProductRecipeStepNo := DSArmBasketInfo.iProductRecipeStepNo + 1;
			END_IF


			IF NOT AR3sbArmPositionCFM[iArmNo,iPickStnNo_ReadInt,4] THEN
			bMoveTop := TRUE;
			ELSE
			bMoveTop := FALSE;
			bStationDrippingTimeST := TRUE;
			END_IF

			IF bStationDrippingTimeST AND tStationDrippingTime.Q THEN
			bStepDelayEn := TRUE;
			END_IF

			IF AR3sbArmPositionCFM[iArmNo,iPickStnNo_ReadInt,4] AND bStationDrippingTimeST AND tStationDrippingTime.Q AND tStepDelay.Q AND NOT bMovingHalt THEN
			bStepDelayEn := FALSE;
			bStationDrippingTimeST := FALSE;
			iPnpStep := 6;
			END_IF

		
		4: (*At Pick Station - Hook*)
		
			IF NOT AR3sbArmPositionCFM[iArmNo,iPickStnNo_ReadInt,3] THEN
		
				IF iPickStnNo_Read = iLdStnID THEN
				bMoveLdHook := TRUE;
				END_IF
		
				IF iPickStnNo_Read = iUldStnID THEN
				bMoveUldHook := TRUE;
				END_IF

				IF iPickStnNo_Read >= 1 AND  iPickStnNo_Read <= iStnQty THEN
				ARbMoveStnHook[iPickStnNo_Read] := TRUE;
				END_IF
		
			ELSE
		
				IF iPickStnNo_Read >= 1 AND  iPickStnNo_Read <= iStnQty THEN
				ARbMoveStnHook[iPickStnNo_Read] := FALSE;
				ELSIF iPickStnNo_Read = iLdStnID THEN
				bMoveLdHook := FALSE;
				ELSIF iPickStnNo_Read = iUldStnID THEN
				bMoveUldHook := FALSE;
				END_IF
		
				bStepDelayEn := TRUE;
		
			END_IF

			IF AR3sbArmPositionCFM[iArmNo,iPickStnNo_ReadInt,3] AND tStepDelay.Q AND NOT bMovingHalt THEN
			bStepDelayEn := FALSE;
			iPnpStep := 5;
			END_IF
		
		
		3: (*Move Vertical Down Pos*)
		
		IF bDownPickCondition THEN
		bDownPickConditionHR := TRUE;
		END_IF

			IF bDownPickConditionHR AND NOT ARbPickMidDownStnEn[iPickStnNo_Read] AND NOT AR3sbArmPositionCFM[iArmNo,iPickStnNo_ReadInt,2] THEN

				IF iPickStnNo_Read = iLdStnID THEN
				bMoveLdDown := TRUE;
				END_IF
		
				IF iPickStnNo_Read = iUldStnID THEN
				bMoveUldDown := TRUE;
				END_IF
		
				IF iPickStnNo_Read >= 1 AND  iPickStnNo_Read <= iStnQty  THEN
				ARbMoveStnDown[iPickStnNo_Read] := TRUE;
				END_IF

			ELSIF bDownPickConditionHR AND ARbPickMidDownStnEn[iPickStnNo_Read] AND NOT AR3sbArmPositionCFM[iArmNo,iPickStnNo_ReadInt,5] THEN

				IF iPickStnNo_Read >= 1 AND  iPickStnNo_Read <= iStnQty  THEN
				ARbMoveStnMidDown[iPickStnNo_Read] := TRUE;
				END_IF

			END_IF

			IF
			(*bDownPickConditionHR AND*) NOT ARbPickMidDownStnEn[iPickStnNo_Read] AND AR3sbArmPositionCFM[iArmNo,iPickStnNo_ReadInt,2]
			OR
			(*bDownPickConditionHR AND*) ARbPickMidDownStnEn[iPickStnNo_Read] AND AR3sbArmPositionCFM[iArmNo,iPickStnNo_ReadInt,5]
			THEN
				IF iPickStnNo_Read >= 1 AND  iPickStnNo_Read <= iStnQty THEN
				ARbMoveStnMidDown[iPickStnNo_Read] := FALSE;
				ARbMoveStnDown[iPickStnNo_Read] := FALSE;
				ELSIF iPickStnNo_Read = iLdStnID THEN
				bMoveLdDown := FALSE;
				ELSIF iPickStnNo_Read = iUldStnID THEN
				bMoveUldDown := FALSE;
				END_IF

				bStepDelayEn := TRUE;

				IF tStepDelay.Q AND NOT bMovingHalt THEN
				bStepDelayEn := FALSE;
				bDownPickConditionHR := FALSE;
				iPnpStep := 4;
				END_IF

			END_IF


		
		
		2: (*Move to Pick Station - Horizontal Unhook Movement*)

			IF NOT AR3sbArmPositionCFM[iArmNo,iPickStnNo_ReadInt,1] THEN
		
				IF iPickStnNo_Read = iLdStnID THEN
				bMoveLdUnhook := TRUE;
				END_IF
		
				IF iPickStnNo_Read = iUldStnID THEN
				bMoveUldUnhook := TRUE;
				END_IF
		
				IF iPickStnNo_Read >= 1 AND  iPickStnNo_Read <= iStnQty THEN
				ARbMoveStnUnhook[iPickStnNo_Read] := TRUE;
				END_IF
		
			ELSE

				IF iPickStnNo_Read >= 1 AND  iPickStnNo_Read <= iStnQty THEN
				ARbMoveStnUnhook[iPickStnNo_Read] := FALSE;
				ELSIF iPickStnNo_Read = iLdStnID THEN
				bMoveLdUnhook := FALSE;
				ELSIF iPickStnNo_Read = iUldStnID THEN
				bMoveUldUnhook := FALSE;
				END_IF
		
				bStepDelayEn := TRUE;
		
			END_IF
		
			IF AR3sbArmPositionCFM[iArmNo,iPickStnNo_ReadInt,1] AND tStepDelay.Q AND NOT bMovingHalt THEN
			bStepDelayEn := FALSE;
			iPnpStep := 3;
			END_IF
		
		
		1: (*Confirm Vertical Top Pos*)
		
			IF NOT AR3sbArmPositionCFM[iArmNo,iCurrentHorzZoneNoint,4] THEN
			bMoveTop := TRUE;
			ELSE
			bMoveTop := FALSE;
			bStepDelayEn := TRUE;
			END_IF
		
			IF AR3sbArmPositionCFM[iArmNo,iCurrentHorzZoneNoint,4] AND tStepDelay.Q AND NOT bMovingHalt THEN
			bStepDelayEn := FALSE;
			iPnpStep := 2;
			END_IF

		0:;







		END_CASE


END_IF

(*Message Display*)

IF NOT bEN THEN
sStatusMessage := 'Arm Not Ready - Homing Required';
ELSIF NOT bPnpStart_Read THEN
sStatusMessage := 'Standby';
END_IF

IF iPnpStep = 1 THEN
sStatusMessage := 'Pnp In Progress - Step 1 - Vertical Up Position';

ELSIF iPnpStep = 2 THEN
sStatusMessage := 'Pnp In Progress - Step 2 - Horizontal Move - Pick Unhook Position';

ELSIF iPnpStep = 3 AND NOT bDownPickCondition THEN
sStatusMessage := 'Pnp In Progress - Step 3 - Waiting Down Pick Condition';

ELSIF iPnpStep = 3 AND bDownPickCondition THEN
sStatusMessage := 'Pnp In Progress - Step 3 - Pick Station Vertical Down Position';

ELSIF iPnpStep = 4 THEN
sStatusMessage := 'Pnp In Progress - Step 4 - Horizontal Move - Pick Hook Position';

ELSIF iPnpStep = 5 AND NOT bStationDrippingTimeST THEN
sStatusMessage := 'Pnp In Progress - Step 5 - Pick Station Vertical Up Position';

ELSIF iPnpStep = 5 AND bStationDrippingTimeST THEN
sStatusMessage := 'Pnp In Progress - Step 5 - Dripping Time Counting';

ELSIF iPnpStep = 6 THEN
sStatusMessage := 'Pnp In Progress - Step 6 - Horizontal Move - Transfer Hook Position';

ELSIF iPnpStep = 7 AND NOT bDownTransferCondition THEN
sStatusMessage := 'Pnp In Progress - Step 7 - Waiting Down Transfer Condition';

ELSIF iPnpStep = 7 AND bDownTransferCondition THEN
sStatusMessage := 'Pnp In Progress - Step 7 - Transfer Station Vertical Down Position';

ELSIF iPnpStep = 8 THEN
sStatusMessage := 'Pnp In Progress - Step 8 - Horizontal Move - Transfer Unhook Position';

ELSIF iPnpStep = 9 THEN
sStatusMessage := 'Pnp In Progress - Step 9 - Transfer Station Vertical Up Position';

ELSIF iPnpStep = 10 THEN
sStatusMessage := 'Pnp Completed';
END_IF

(*Arm Pnp Completed*)
IF bPnpCompleted THEN
	ARiStnNoToCalledArm_Uni[iArmNo] 					:= 0;
	ARDSGnrFeedArmPnpParameter_Uni[iArmNo] 		:= DSEmptyGnrCalledArmPnpParameter;
END_IF


(*Arm Ready Bit*)
IF bEN AND NOT bPnpBusy AND NOT bPnpStart_Read THEN
bArmReady	:= TRUE;
ELSE
bArmReady 	:= FALSE;
END_IF


(*Reset Output*)
IF NOT bEN OR bReset OR bPnpStart_Read_FE.Q THEN

	bPnpCompleted 									:= FALSE;
	bPnpBusy										:= FALSE;
	bMoveTop										:= FALSE;
	bMoveLdDown									:= FALSE;
	bMoveUldDown									:= FALSE;
	bMoveLdHook									:= FALSE;
	bMoveLdUnhook									:= FALSE;
	bMoveUldHook									:= FALSE;
	bMoveUldUnhook									:= FALSE;
	iPnpStep											:= 0;
	bDownPickConditionHR 							:= FALSE;
	bDownTransferConditionHR 						:= FALSE;
	bStepDelayEn 									:= FALSE;
	ARiStnNoToCalledArm_Uni[iArmNo] 					:= 0;
	ARDSGnrFeedArmPnpParameter_Uni[iArmNo] 		:= DSEmptyGnrCalledArmPnpParameter;

	iResetFL := 1;
	FOR iResetFL := 1 TO iStnQty DO
		IF iResetFL >= 1 AND iResetFL <= iStnQty THEN
			ARbMoveStnMidDown[iResetFL]			:=	FALSE;
			ARbMoveStnDown[iResetFL]				:=	FALSE;
			ARbMoveStnHook[iResetFL]				:=	FALSE;
			ARbMoveStnUnhook[iResetFL]				:=	FALSE;
		END_IF
	END_FOR

END_IF

END_FUNCTION_BLOCK

// ---- FBs/B_JKS_CustomFB/fbArmCtrlFolder/fbAxisPosCtrl.TcPOU
FUNCTION_BLOCK fbAxisPosCtrl
VAR_INPUT

	bAxis1EN : BOOL;
	bAxis2EN : BOOL;
	bAxis3EN : BOOL;
	bAxis4EN : BOOL;

	bPosStart : BOOL;
	bHomingRdy : BOOL;
	wTargetPosNum : DWORD;
	lrFixVelo : LREAL;
	lrFixAcc : LREAL;
	lrFixDcc : LREAL;
	lrCurrentServoPos : LREAL;
	lrPos1 : LREAL;
	lrPos2 : LREAL;
	lrPos3 : LREAL;
	lrPos4 : LREAL;
	lrPos5 : LREAL;
	lrPos6 : LREAL;
	lrPos7 : LREAL;
	lrPos8 : LREAL;
	lrPos9 : LREAL;
	lrPos10 : LREAL;
	lrPos11 : LREAL;
	lrPos12 : LREAL;
	lrPos13 : LREAL;
	lrPos14 : LREAL;
	lrPos15 : LREAL;
	lrPos16 : LREAL;
	lrPos17 : LREAL;
	lrPos18 : LREAL;
	lrPos19 : LREAL;
	lrPos20 : LREAL;
	lrPos21 : LREAL;
	lrPos22 : LREAL;
	lrPos23 : LREAL;
	lrPos24 : LREAL;
	lrPos25 : LREAL;

END_VAR
VAR_IN_OUT
	Arm1HorzReady: BOOL;
	Arm1VertReady: BOOL;
	Arm1Vert : axis_ref;
	Arm1Horz : axis_ref;
END_VAR

VAR_OUTPUT

	AxisStopEn : BOOL;

END_VAR
VAR
	Stoptimer: TON;
	AxisStopbit: BOOL;
	TimerMove: TON;
	BlockStartBit: BOOL;
	PosSV: LREAL;
	Move1: BOOL;
	Move2: BOOL;
	Move3: BOOL;
	Move4: BOOL;
	Move5: BOOL;
	Move6: BOOL;
	Move7: BOOL;
	Move8: BOOL;
	Move9: BOOL;
	Move10: BOOL;
	Move11: BOOL;
	Move12: BOOL;
	Move13: BOOL;
	Move14: BOOL;
	Move15: BOOL;
	Move16: BOOL;
	Move17: BOOL;
	Move18: BOOL;
	Move19: BOOL;
	Move20: BOOL;
	Move21: BOOL;
	Move22: BOOL;
	Move23: BOOL;
	Move24: BOOL;
	Move25: BOOL;
	Halt1: MC_Halt;
	Halt2: MC_Halt;
	Halt3: MC_Halt;
	Halt4: MC_Halt;
	ArmMoveTostation2: MC_MoveAbsolute;
	ArmMoveTostation: MC_MoveAbsolute;
	ArmMoveTostation3: MC_MoveAbsolute;
	ArmMoveTostation4: MC_MoveAbsolute;
	AxisStopEn1: BOOL;
	AxisStopEn2: BOOL;
	AxisStopEn3: BOOL;
	AxisStopEn4: BOOL;
	Arm1VertReadStatus: MC_ReadStatus;
	Arm1HorzReadStatus: MC_ReadStatus;
END_VAR
VAR // added by the converter: edge detectors and wires of the graphical bodies
    _w1, _w2, _w3, _w4, _w5, _w6, _w7, _w8, _w9, _w10, _w11, _w12, _w13, _w14, _w15, _w16, _w17, _w18, _w19, _w20, _w21, _w22, _w23, _w24, _w25 : LREAL;
END_VAR

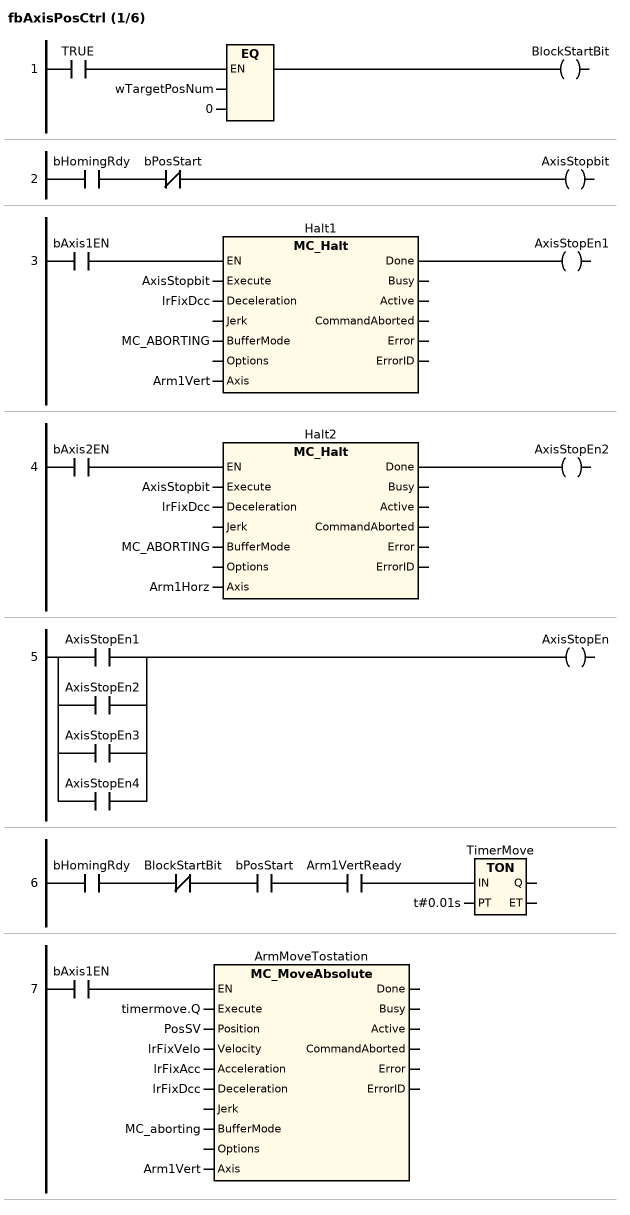
// NETWORK 1
BlockStartBit := wTargetPosNum = 0;

// NETWORK 2
AxisStopbit := bHomingRdy AND NOT bPosStart;

// NETWORK 3
IF bAxis1EN THEN
    Halt1(Execute := AxisStopbit, Deceleration := lrFixDcc, BufferMode := MC_ABORTING, Axis := Arm1Vert); // MC_Halt
END_IF
AxisStopEn1 := Halt1.Done;

// NETWORK 4
IF bAxis2EN THEN
    Halt2(Execute := AxisStopbit, Deceleration := lrFixDcc, BufferMode := MC_ABORTING, Axis := Arm1Horz); // MC_Halt
END_IF
AxisStopEn2 := Halt2.Done;

// NETWORK 5
AxisStopEn := AxisStopEn1 OR AxisStopEn2 OR AxisStopEn3 OR AxisStopEn4;

// NETWORK 6
TimerMove(IN := bHomingRdy AND NOT BlockStartBit AND bPosStart AND Arm1VertReady, PT := t#0.01s); // TON

// NETWORK 7
IF bAxis1EN THEN
    ArmMoveTostation(
        Execute := timermove.Q,
        Position := PosSV,
        Velocity := lrFixVelo,
        Acceleration := lrFixAcc,
        Deceleration := lrFixDcc,
        BufferMode := MC_aborting,
        Axis := Arm1Vert); // MC_MoveAbsolute
END_IF

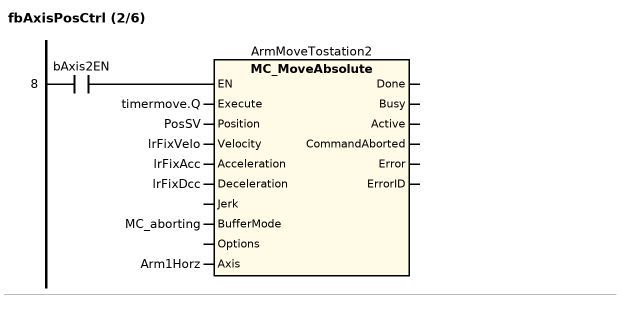
// NETWORK 8
IF bAxis2EN THEN
    ArmMoveTostation2(
        Execute := timermove.Q,
        Position := PosSV,
        Velocity := lrFixVelo,
        Acceleration := lrFixAcc,
        Deceleration := lrFixDcc,
        BufferMode := MC_aborting,
        Axis := Arm1Horz); // MC_MoveAbsolute
END_IF

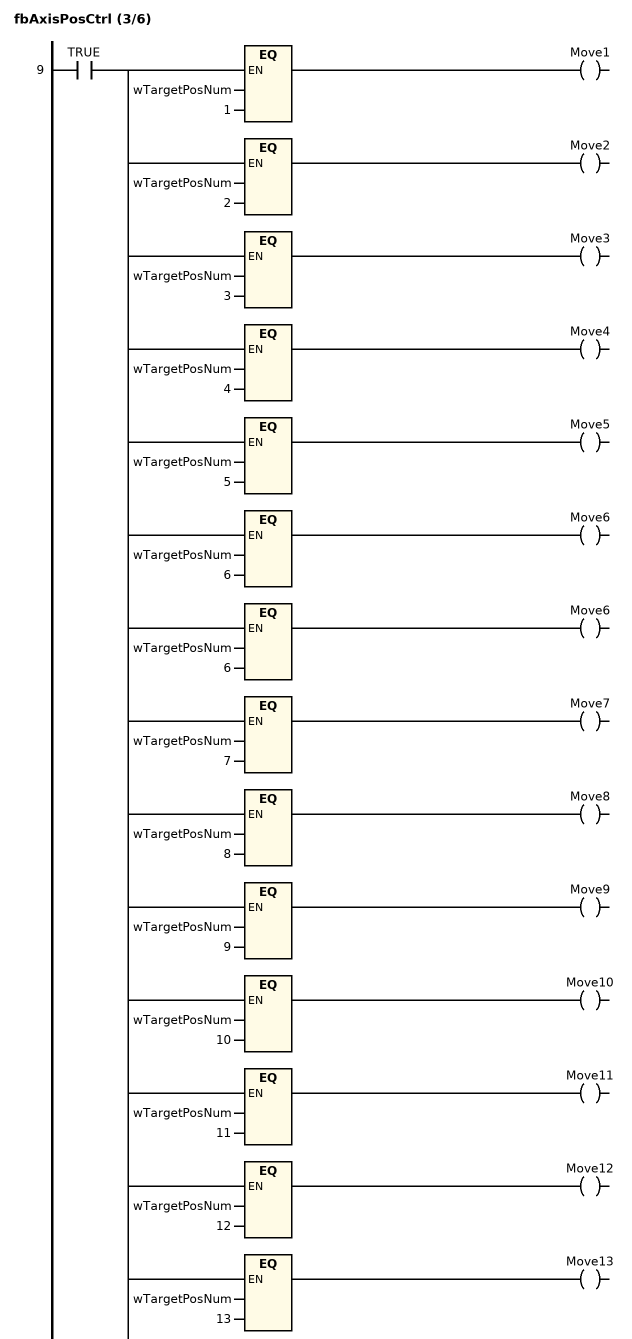
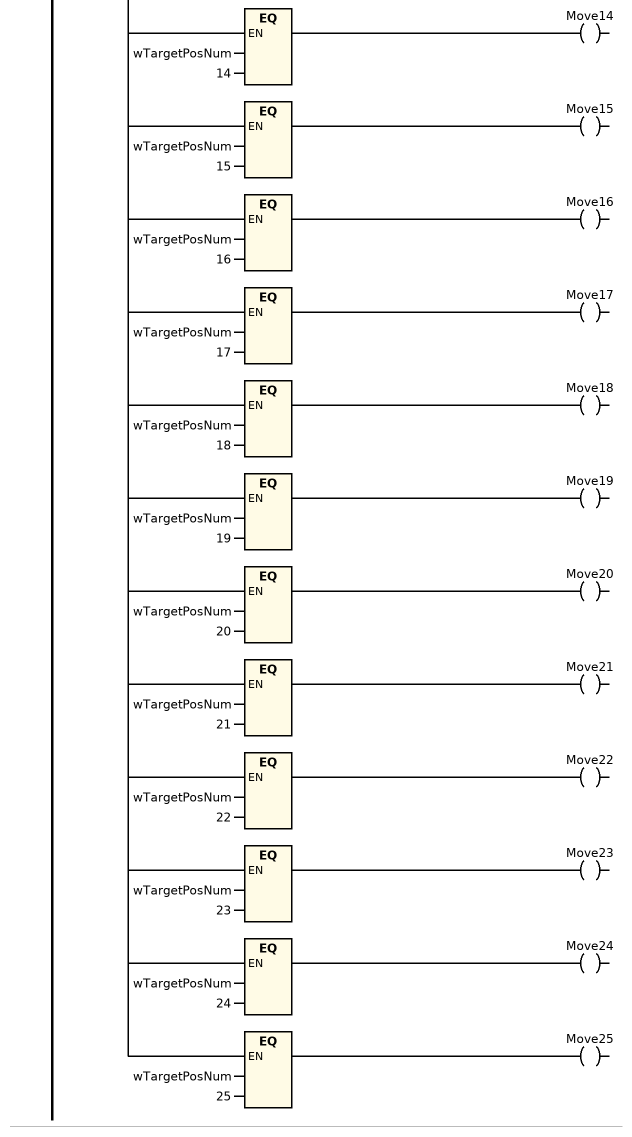
// NETWORK 9
Move1 := wTargetPosNum = 1;
Move2 := wTargetPosNum = 2;
Move3 := wTargetPosNum = 3;
Move4 := wTargetPosNum = 4;
Move5 := wTargetPosNum = 5;
Move6 := wTargetPosNum = 6;
Move6 := wTargetPosNum = 6;
Move7 := wTargetPosNum = 7;
Move8 := wTargetPosNum = 8;
Move9 := wTargetPosNum = 9;
Move10 := wTargetPosNum = 10;
Move11 := wTargetPosNum = 11;
Move12 := wTargetPosNum = 12;
Move13 := wTargetPosNum = 13;
Move14 := wTargetPosNum = 14;
Move15 := wTargetPosNum = 15;
Move16 := wTargetPosNum = 16;
Move17 := wTargetPosNum = 17;
Move18 := wTargetPosNum = 18;
Move19 := wTargetPosNum = 19;
Move20 := wTargetPosNum = 20;
Move21 := wTargetPosNum = 21;
Move22 := wTargetPosNum = 22;
Move23 := wTargetPosNum = 23;
Move24 := wTargetPosNum = 24;
Move25 := wTargetPosNum = 25;

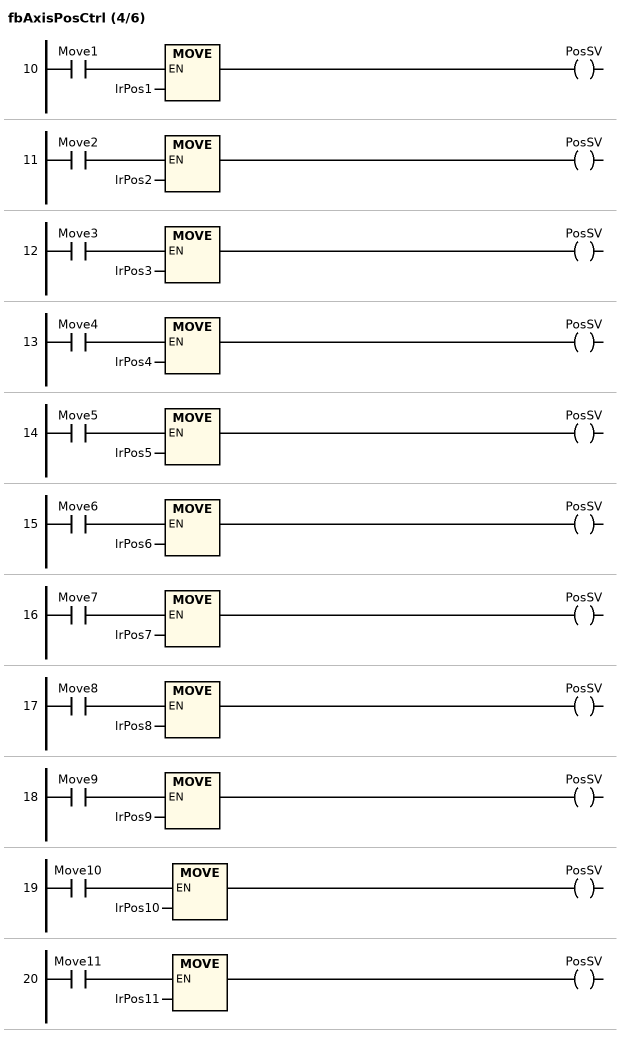
// NETWORK 10
IF Move1 THEN _w1 := lrPos1; END_IF
PosSV := _w1;

// NETWORK 11
IF Move2 THEN _w2 := lrPos2; END_IF
PosSV := _w2;

// NETWORK 12
IF Move3 THEN _w3 := lrPos3; END_IF
PosSV := _w3;

// NETWORK 13
IF Move4 THEN _w4 := lrPos4; END_IF
PosSV := _w4;

// NETWORK 14
IF Move5 THEN _w5 := lrPos5; END_IF
PosSV := _w5;

// NETWORK 15
IF Move6 THEN _w6 := lrPos6; END_IF
PosSV := _w6;

// NETWORK 16
IF Move7 THEN _w7 := lrPos7; END_IF
PosSV := _w7;

// NETWORK 17
IF Move8 THEN _w8 := lrPos8; END_IF
PosSV := _w8;

// NETWORK 18
IF Move9 THEN _w9 := lrPos9; END_IF
PosSV := _w9;

// NETWORK 19
IF Move10 THEN _w10 := lrPos10; END_IF
PosSV := _w10;

// NETWORK 20
IF Move11 THEN _w11 := lrPos11; END_IF
PosSV := _w11;

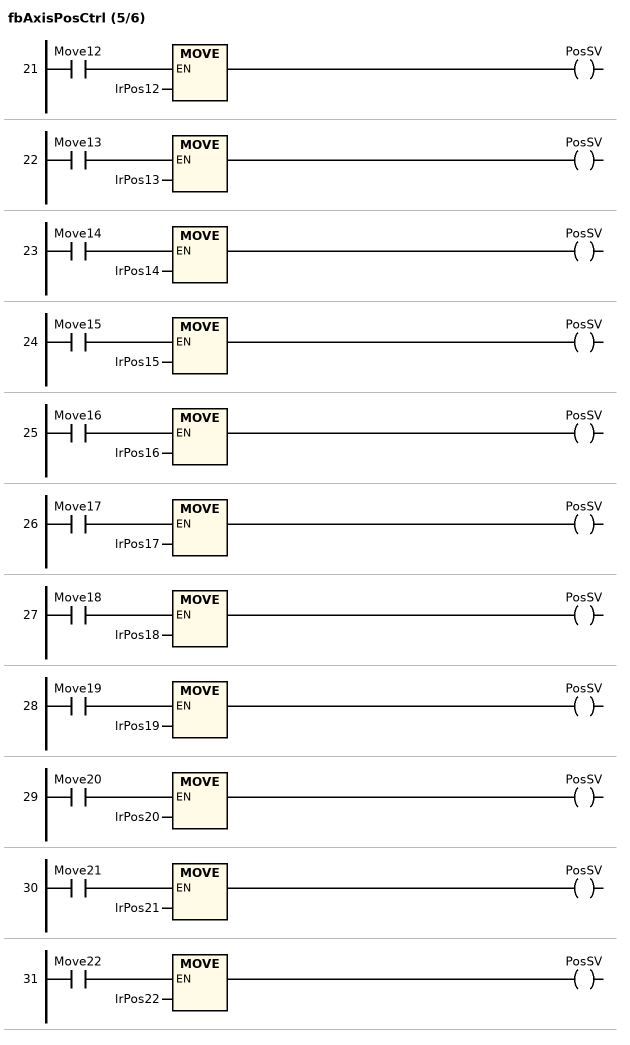
// NETWORK 21
IF Move12 THEN _w12 := lrPos12; END_IF
PosSV := _w12;

// NETWORK 22
IF Move13 THEN _w13 := lrPos13; END_IF
PosSV := _w13;

// NETWORK 23
IF Move14 THEN _w14 := lrPos14; END_IF
PosSV := _w14;

// NETWORK 24
IF Move15 THEN _w15 := lrPos15; END_IF
PosSV := _w15;

// NETWORK 25
IF Move16 THEN _w16 := lrPos16; END_IF
PosSV := _w16;

// NETWORK 26
IF Move17 THEN _w17 := lrPos17; END_IF
PosSV := _w17;

// NETWORK 27
IF Move18 THEN _w18 := lrPos18; END_IF
PosSV := _w18;

// NETWORK 28
IF Move19 THEN _w19 := lrPos19; END_IF
PosSV := _w19;

// NETWORK 29
IF Move20 THEN _w20 := lrPos20; END_IF
PosSV := _w20;

// NETWORK 30
IF Move21 THEN _w21 := lrPos21; END_IF
PosSV := _w21;

// NETWORK 31
IF Move22 THEN _w22 := lrPos22; END_IF
PosSV := _w22;

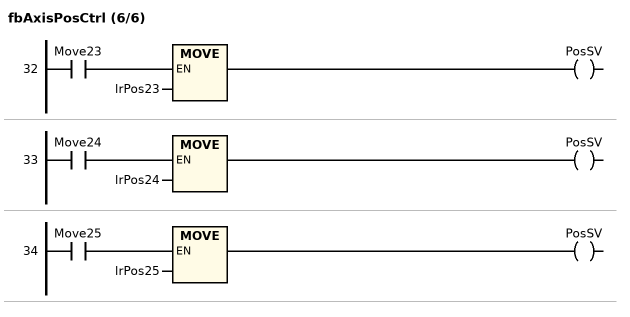
// NETWORK 32
IF Move23 THEN _w23 := lrPos23; END_IF
PosSV := _w23;

// NETWORK 33
IF Move24 THEN _w24 := lrPos24; END_IF
PosSV := _w24;

// NETWORK 34
IF Move25 THEN _w25 := lrPos25; END_IF
PosSV := _w25;

END_FUNCTION_BLOCK

// ---- FBs/B_JKS_CustomFB/fbArmCtrlFolder/fbGenerateArmPickTransferBit.TcPOU
FUNCTION_BLOCK fbGenerateArmPickTransferBit
VAR_INPUT
	iPickStationNo : INT;
	iTransferStationNo : INT;
	bArmBusy	: BOOL;
END_VAR
VAR_OUTPUT
	bArmPickLd : BOOL;
	bArmPickUld : BOOL;
	ARbArmPickStn : ARRAY [1..iStnQty] OF BOOL;
	bArmTransferLd : BOOL;
	bArmTransferUld : BOOL;
	ARbArmTransferStn : ARRAY [1..iStnQty] OF BOOL;

END_VAR
VAR
	iPickStnFL: INT;
	iClearPickStnFL: INT;
	iTransferStnFL: INT;
	iClearTransferStnFL: INT;
END_VAR

IF bArmBusy AND iPickStationNo = iLdStnID THEN
bArmPickLd := TRUE;
ELSIF bArmBusy AND  iPickStationNo = iUldStnID THEN
bArmPickUld := TRUE;
ELSIF bArmBusy AND  iPickStationNo >= 1 AND iPickStationNo <= iStnQty THEN
iPickStnFL := 1;
	FOR iPickStnFL := 1 TO iStnQty DO
		IF iPickStnFL >= 1 AND iPickStnFL <= iStnQty THEN
			IF iPickStationNo = iPickStnFL THEN
				ARbArmPickStn[iPickStnFL] := TRUE;
			END_IF
		END_IF
	END_FOR
ELSE
bArmPickLd := FALSE;
bArmPickUld := FALSE;
iClearPickStnFL := 1;
	FOR iClearPickStnFL := 1 TO iStnQty DO
		IF iClearPickStnFL >= 1 AND iClearPickStnFL <= iStnQty THEN
				ARbArmPickStn[iClearPickStnFL] := FALSE;
		END_IF
	END_FOR
END_IF

IF bArmBusy AND  iTransferStationNo = iLdStnID THEN
bArmTransferLd := TRUE;
ELSIF bArmBusy AND iTransferStationNo = iUldStnID THEN
bArmTransferUld := TRUE;
ELSIF bArmBusy AND iTransferStationNo >= 1 AND iTransferStationNo <= iStnQty THEN
iTransferStnFL := 1;
	FOR iTransferStnFL := 1 TO iStnQty DO
		IF iTransferStnFL >= 1 AND iTransferStnFL <= iStnQty THEN
			IF iTransferStationNo = iTransferStnFL THEN
				ARbArmTransferStn[iTransferStnFL] := TRUE;
			END_IF
		END_IF
	END_FOR
ELSE
bArmTransferLd := FALSE;
bArmTransferUld := FALSE;
iClearTransferStnFL := 1;
	FOR iClearTransferStnFL := 1 TO iStnQty DO
		IF iClearTransferStnFL >= 1 AND iClearTransferStnFL <= iStnQty THEN
				ARbArmTransferStn[iClearTransferStnFL] := FALSE;
		END_IF
	END_FOR
END_IF

END_FUNCTION_BLOCK

// ---- FBs/B_JKS_CustomFB/fbArmCtrlFolder/fbInverterHorzHome.TcPOU
FUNCTION_BLOCK fbInverterHorzHome
VAR_INPUT
	bExecute	: BOOL;
	bEstop		: BOOL;
	bHomeFor	: BOOL;
	bHomeRev	: BOOL;
	bHomeSenser	: BOOL;
	bOTsensor1		: BOOL;
	bOTsensor2		: BOOL;
	bReset			: BOOL;
	i1stRPM			: INT;
	i2ndRPM			: INT;
	rInverterRatio		: REAL;
	EncoderRatio		: LREAL;

END_VAR
VAR_OUTPUT
	bDone		: BOOL;
	bBusy		: BOOL;
	bError		: BOOL;
	bMovForBit	: BOOL;
	bMovRevBit	: BOOL;
	bMovFor2ndBit	: BOOL;
	bMovRev2ndBit	: BOOL;
	bMovFor3rdBit	: BOOL;
	bMovRev3rdBit	: BOOL;
	lrActualPosReference	: LREAL;

END_VAR
VAR_IN_OUT

	iHomeHzout	: INT;
	Axis1		: axis_ref;

END_VAR
VAR
	MCRAP1: MC_ReadActualPosition;
	PowerRelay: TON;
	ArmMovActualPos: LREAL;
	RTRIG1: R_TRIG;
	Move2Home: BOOL;
	HomingStop: BOOL;
	Conv1: AM_InverterConversionHz;
	Conv2: AM_InverterConversionHz;
	CMP1: fbServoPosCmp;
	ArmReachHome: BOOL;
	Conv3: AM_InverterConversionHz;
	Conv4: AM_InverterConversionHz;
	MoveAwayHome: BOOL;
	Conv5: AM_InverterConversionHz;
	Conv6: AM_InverterConversionHz;
	HomingStep1: BOOL;
	MCSPOS1: MC_SetPosition;
	SetPosDone: BOOL;
	TON2: TON;
	T1: TON;
	T2: TON;
	HomeSensorTriggerBit: BOOL;
	HomingStep2: BOOL;
	OTstop: BOOL;
	TRIG1: R_TRIG;
	TRIG2: R_TRIG;
	RTRIG2: R_TRIG;
	i1stRPMTemp: INT;
	i2ndRPMTemp: INT;
	LrPosBeforeConvert: LREAL;
	TON10: TON;
END_VAR

VAR PERSISTENT

	HorzArmPos : LREAL;

END_VAR
VAR // added by the converter: edge detectors and wires of the graphical bodies
    _w1, _w2 : INT;
    _w3 : LREAL;
END_VAR

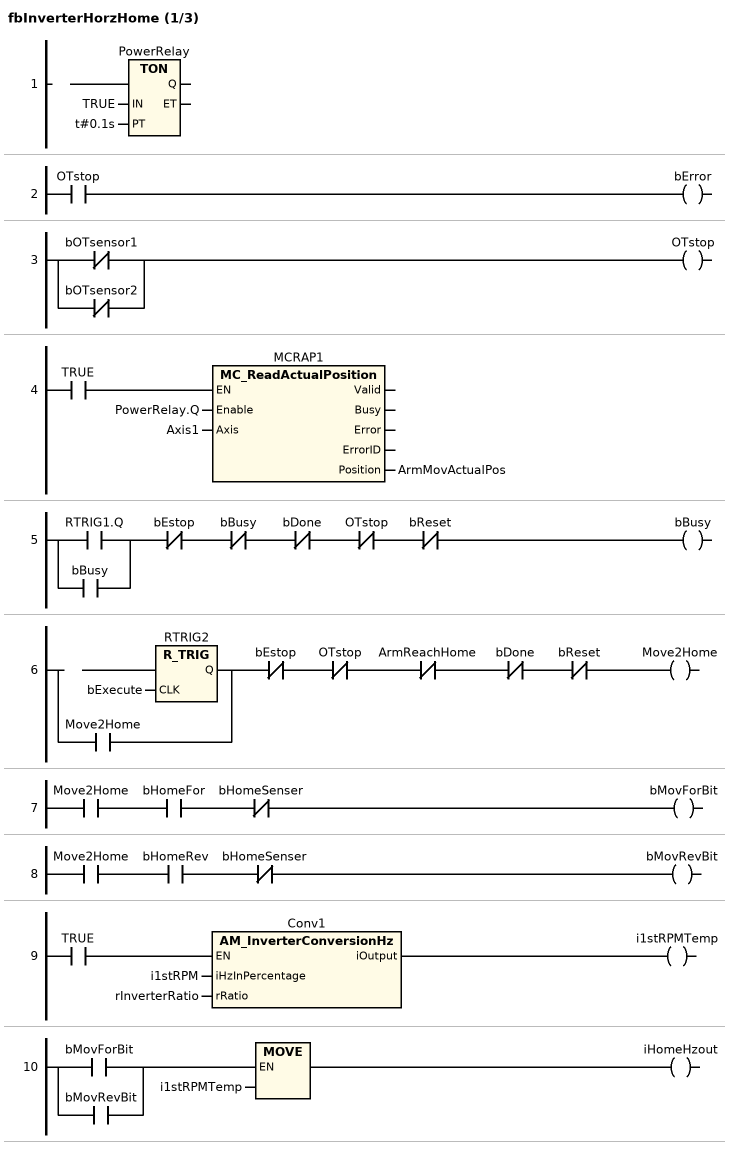
// NETWORK 1
PowerRelay(IN := TRUE, PT := t#0.1s); // TON

// NETWORK 2
bError := OTstop;

// NETWORK 3
OTstop := NOT bOTsensor1 OR NOT bOTsensor2;

// NETWORK 4
MCRAP1(Enable := PowerRelay.Q, Axis := Axis1, Position => ArmMovActualPos); // MC_ReadActualPosition

// NETWORK 5
bBusy := (RTRIG1.Q OR bBusy) AND NOT bEstop AND NOT bBusy AND NOT bDone AND NOT OTstop AND NOT bReset;

// NETWORK 6
RTRIG2(CLK := bExecute); // R_TRIG
Move2Home := (RTRIG2.Q OR Move2Home) AND NOT bEstop AND NOT OTstop AND NOT ArmReachHome AND NOT bDone AND NOT bReset;

// NETWORK 7
bMovForBit := Move2Home AND bHomeFor AND NOT bHomeSenser;

// NETWORK 8
bMovRevBit := Move2Home AND bHomeRev AND NOT bHomeSenser;

// NETWORK 9
Conv1(iHzInPercentage := i1stRPM, rRatio := rInverterRatio); // AM_InverterConversionHz
i1stRPMTemp := Conv1.iOutput;

// NETWORK 10
IF bMovForBit OR bMovRevBit THEN _w1 := i1stRPMTemp; END_IF
iHomeHzout := _w1;

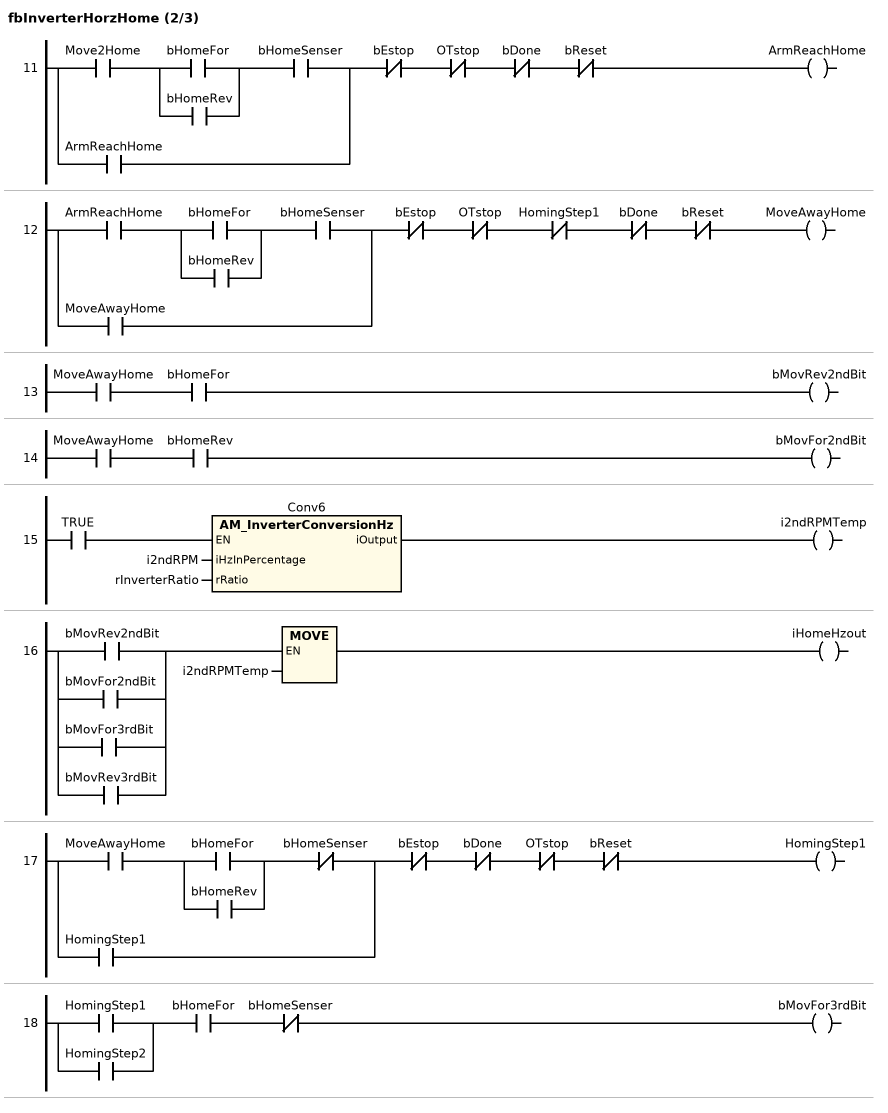
// NETWORK 11
ArmReachHome := ((Move2Home AND (bHomeFor OR bHomeRev)) AND bHomeSenser OR ArmReachHome) AND NOT bEstop AND NOT OTstop AND NOT bDone AND NOT bReset;

// NETWORK 12
MoveAwayHome := ((ArmReachHome AND (bHomeFor OR bHomeRev)) AND bHomeSenser OR MoveAwayHome) AND NOT bEstop AND NOT OTstop AND NOT HomingStep1 AND NOT bDone AND NOT bReset;

// NETWORK 13
bMovRev2ndBit := MoveAwayHome AND bHomeFor;

// NETWORK 14
bMovFor2ndBit := MoveAwayHome AND bHomeRev;

// NETWORK 15
Conv6(iHzInPercentage := i2ndRPM, rRatio := rInverterRatio); // AM_InverterConversionHz
i2ndRPMTemp := Conv6.iOutput;

// NETWORK 16
IF bMovRev2ndBit OR bMovFor2ndBit OR bMovFor3rdBit OR bMovRev3rdBit THEN _w2 := i2ndRPMTemp; END_IF
iHomeHzout := _w2;

// NETWORK 17
HomingStep1 := ((MoveAwayHome AND (bHomeFor OR bHomeRev)) AND NOT bHomeSenser OR HomingStep1) AND NOT bEstop AND NOT bDone AND NOT OTstop AND NOT bReset;

// NETWORK 18
bMovFor3rdBit := (HomingStep1 OR HomingStep2) AND bHomeFor AND NOT bHomeSenser;

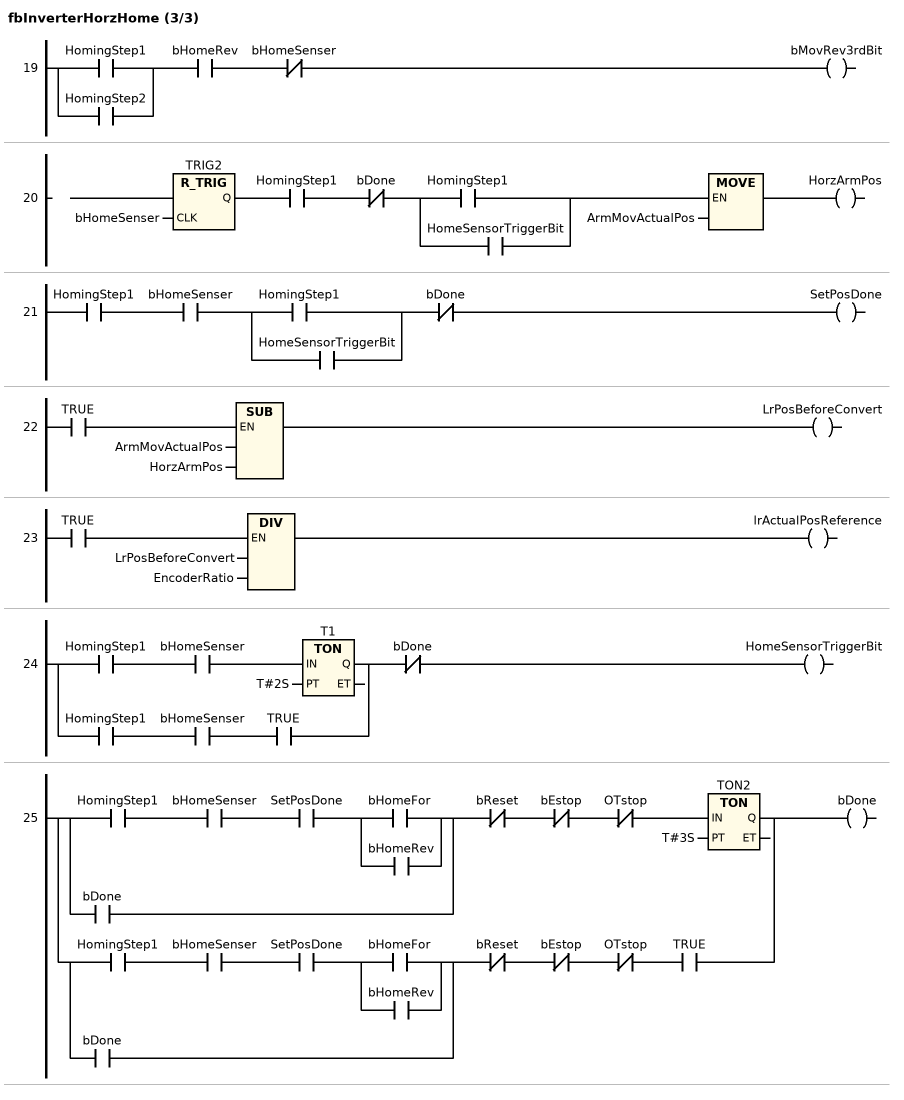
// NETWORK 19
bMovRev3rdBit := (HomingStep1 OR HomingStep2) AND bHomeRev AND NOT bHomeSenser;

// NETWORK 20
TRIG2(CLK := bHomeSenser); // R_TRIG
IF TRIG2.Q AND HomingStep1 AND NOT bDone AND (HomingStep1 OR HomeSensorTriggerBit) THEN
    _w3 := ArmMovActualPos;
END_IF
HorzArmPos := _w3;

// NETWORK 21
SetPosDone := (HomingStep1 AND bHomeSenser AND (HomingStep1 OR HomeSensorTriggerBit)) AND NOT bDone;

// NETWORK 22
LrPosBeforeConvert := ArmMovActualPos - HorzArmPos;

// NETWORK 23
lrActualPosReference := LrPosBeforeConvert / EncoderRatio;

// NETWORK 24
T1(IN := HomingStep1 AND bHomeSenser, PT := T#2S); // TON
HomeSensorTriggerBit := (T1.Q OR (HomingStep1 AND bHomeSenser) AND TRUE) AND NOT bDone;

// NETWORK 25
TON2(IN := (HomingStep1 AND bHomeSenser AND SetPosDone AND (bHomeFor OR bHomeRev) OR bDone) AND NOT bReset AND NOT bEstop AND NOT OTstop, PT := T#3S); // TON
bDone := TON2.Q OR ((HomingStep1 AND bHomeSenser AND SetPosDone AND (bHomeFor OR bHomeRev) OR bDone) AND NOT bReset AND NOT bEstop AND NOT OTstop) AND TRUE;

END_FUNCTION_BLOCK

// ---- FBs/B_JKS_CustomFB/fbArmCtrlFolder/fbInverterJogCtrl.TcPOU
FUNCTION_BLOCK fbInverterJogCtrl
VAR_INPUT
	bEnable			: BOOL;
	bEmergencyStop	: BOOL;
	bLeftOT			: BOOL;
	bRightOT		: BOOL;
	bArmJogFor		: BOOL;
	bArmJogRev		: BOOL;
	iJogRPM		: INT;
	rRatio			: REAL;

END_VAR
VAR_OUTPUT
	bMoveForFlag	: BOOL;
	bMoveRevFlag	: BOOL;
END_VAR

VAR_IN_OUT
	iMoveRPM		: INT;

END_VAR
VAR
	LeftOtAlarm: BOOL;
	RightOtAlarm: BOOL;
	JogForFb: AM_InverterConversionHz;
	iMoveRPMTemp: INT;
END_VAR
VAR // added by the converter: edge detectors and wires of the graphical bodies
    _w1, _w2 : INT;
END_VAR

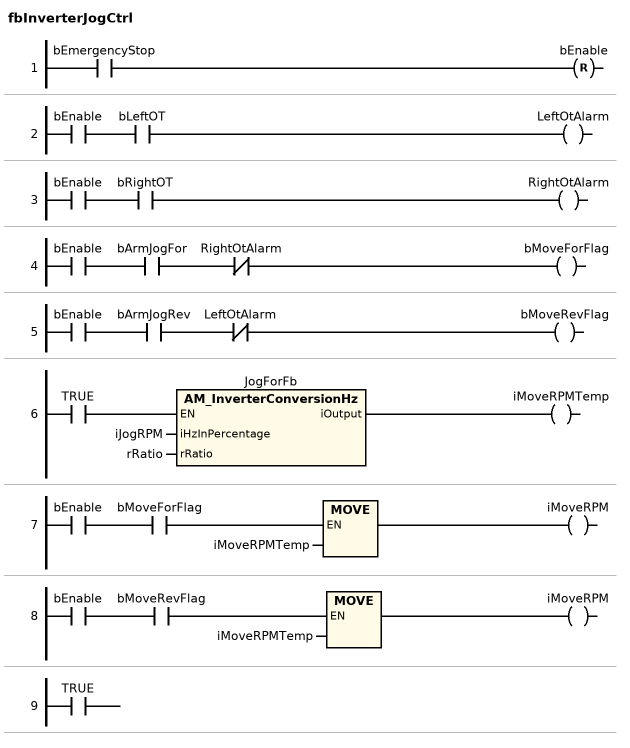
// NETWORK 1
bEnable R= bEmergencyStop;

// NETWORK 2
LeftOtAlarm := bEnable AND bLeftOT;

// NETWORK 3
RightOtAlarm := bEnable AND bRightOT;

// NETWORK 4
bMoveForFlag := bEnable AND bArmJogFor AND NOT RightOtAlarm;

// NETWORK 5
bMoveRevFlag := bEnable AND bArmJogRev AND NOT LeftOtAlarm;

// NETWORK 6
JogForFb(iHzInPercentage := iJogRPM, rRatio := rRatio); // AM_InverterConversionHz
iMoveRPMTemp := JogForFb.iOutput;

// NETWORK 7
IF bEnable AND bMoveForFlag THEN _w1 := iMoveRPMTemp; END_IF
iMoveRPM := _w1;

// NETWORK 8
IF bEnable AND bMoveRevFlag THEN _w2 := iMoveRPMTemp; END_IF
iMoveRPM := _w2;

// NETWORK 9

END_FUNCTION_BLOCK

// ---- FBs/B_JKS_CustomFB/fbArmCtrlFolder/fbInverterPosCtrl.TcPOU
FUNCTION_BLOCK fbInverterPosCtrl
VAR_INPUT
	bHomingRdy		:	BOOL;
	bPosStart		:	BOOL;
	dTargetPosNum	:	DINT;
	i1stRPMfix		:	INT;
	i2ndRPMfix		:	INT;
	i2ndSpdRangefix	:	INT;
	iOffSetRangeFix	:	INT;
	iRatioFix			:	REAL;
	lrActualPosition	:	LREAL;

	iPos1			:	INT;
	iPos2			:	INT;
	iPos3			:	INT;
	iPos4			:	INT;
	iPos5			:	INT;
	iPos6			:	INT;
	iPos7			:	INT;
	iPos8			:	INT;
	iPos9			:	INT;
	iPos10			:	INT;
	iPos11			:	INT;
	iPos12			:	INT;
	iPos13			:	INT;
	iPos14			:	INT;
	iPos15			:	INT;
	iPos16			:	INT;
	iPos17			:	INT;
	iPos18			:	INT;
	iPos19			:	INT;
	iPos20			:	INT;


END_VAR
VAR_OUTPUT
	bMoveDone		:	BOOL;
	bMoveFor		: 	BOOL;
	bMoveRev		:	BOOL;
	iTargetPos		:	INT ;

END_VAR
VAR_IN_OUT
	iSpdOut			:	INT;
	PosSv			:	INT;

END_VAR
VAR

	Move_1: AM_MoveAbsolute;
	Move1: BOOL;
	Move2: BOOL;
	Move3: BOOL;
	Move4: BOOL;
	Move5: BOOL;
	Move6: BOOL;
	Move7: BOOL;
	Move8: BOOL;
	Move9: BOOL;
	Move10: BOOL;
	Move11: BOOL;
	Move12: BOOL;
	Move13: BOOL;
	Move14: BOOL;
	Move15: BOOL;
	Move16: BOOL;
	Move17: BOOL;
	Move18: BOOL;
	Move19: BOOL;
	Move20: BOOL;


	ArmMoveStart: BOOL;
	iSpdOutTemp: INT;
	FB: fbArmMoveInterLock;

	ArmMoveEn: BOOL;
	TON1: TON;
	bSpeedNormalEn: BOOL;
	iSlowSpeedRange: INT;

	iDccTime		:	INT := 5;
	iDccStep			:	INT := 2;
END_VAR
VAR // added by the converter: edge detectors and wires of the graphical bodies
    _w1, _w3, _w4, _w5, _w6, _w7, _w8, _w9, _w10, _w11, _w12, _w13, _w14, _w15, _w16, _w17, _w18, _w19, _w20, _w21, _w22 : INT;
    _w2 : ANY;
END_VAR

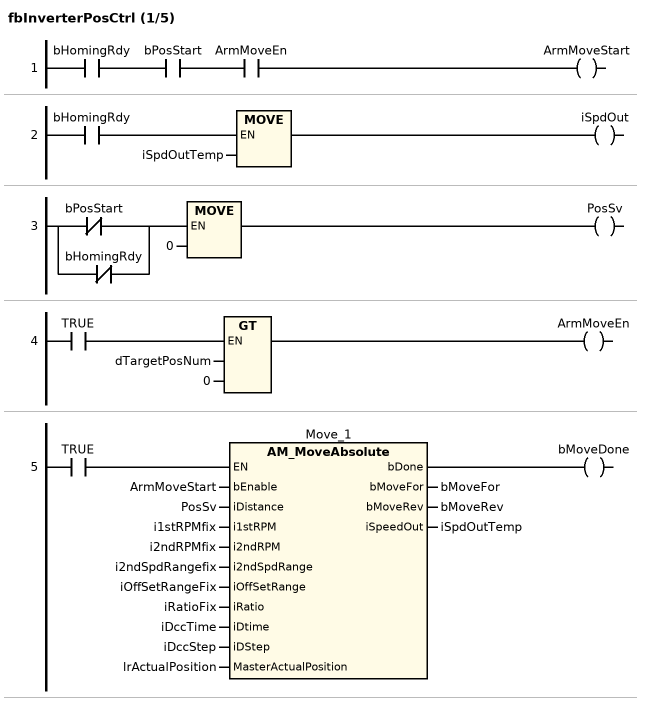
// NETWORK 1
ArmMoveStart := bHomingRdy AND bPosStart AND ArmMoveEn;

// NETWORK 2
IF bHomingRdy THEN _w1 := iSpdOutTemp; END_IF
iSpdOut := _w1;

// NETWORK 3
IF NOT bPosStart OR NOT bHomingRdy THEN _w2 := 0; END_IF
PosSv := _w2;

// NETWORK 4
ArmMoveEn := dTargetPosNum > 0;

// NETWORK 5
Move_1(
    bEnable := ArmMoveStart,
    iDistance := PosSv,
    i1stRPM := i1stRPMfix,
    i2ndRPM := i2ndRPMfix,
    i2ndSpdRange := i2ndSpdRangefix,
    iOffSetRange := iOffSetRangeFix,
    iRatio := iRatioFix,
    iDtime := iDccTime,
    iDStep := iDccStep,
    MasterActualPosition := lrActualPosition,
    bMoveFor => bMoveFor,
    bMoveRev => bMoveRev,
    iSpeedOut => iSpdOutTemp); // AM_MoveAbsolute
bMoveDone := Move_1.bDone;

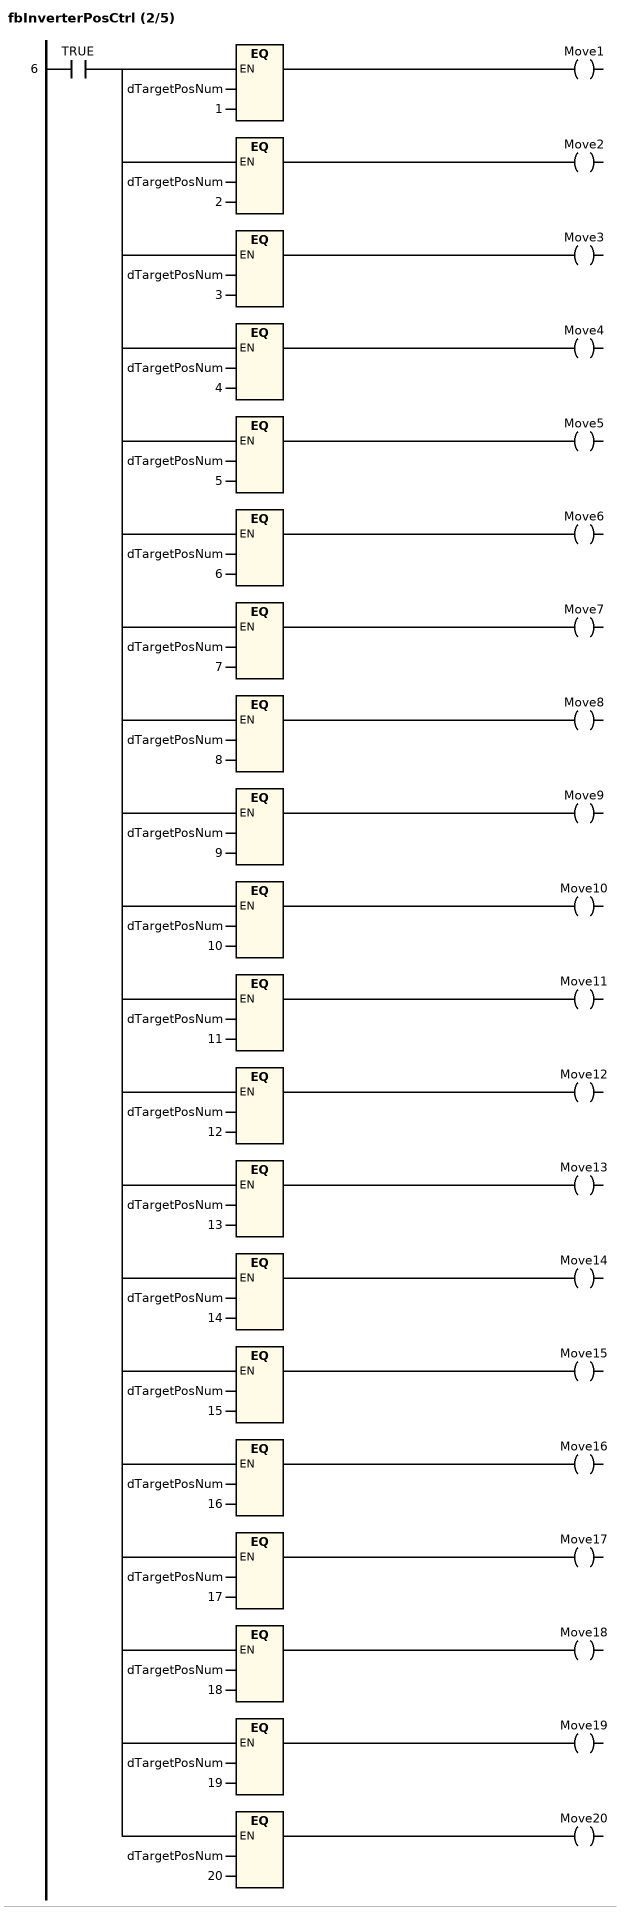
// NETWORK 6
Move1 := dTargetPosNum = 1;
Move2 := dTargetPosNum = 2;
Move3 := dTargetPosNum = 3;
Move4 := dTargetPosNum = 4;
Move5 := dTargetPosNum = 5;
Move6 := dTargetPosNum = 6;
Move7 := dTargetPosNum = 7;
Move8 := dTargetPosNum = 8;
Move9 := dTargetPosNum = 9;
Move10 := dTargetPosNum = 10;
Move11 := dTargetPosNum = 11;
Move12 := dTargetPosNum = 12;
Move13 := dTargetPosNum = 13;
Move14 := dTargetPosNum = 14;
Move15 := dTargetPosNum = 15;
Move16 := dTargetPosNum = 16;
Move17 := dTargetPosNum = 17;
Move18 := dTargetPosNum = 18;
Move19 := dTargetPosNum = 19;
Move20 := dTargetPosNum = 20;

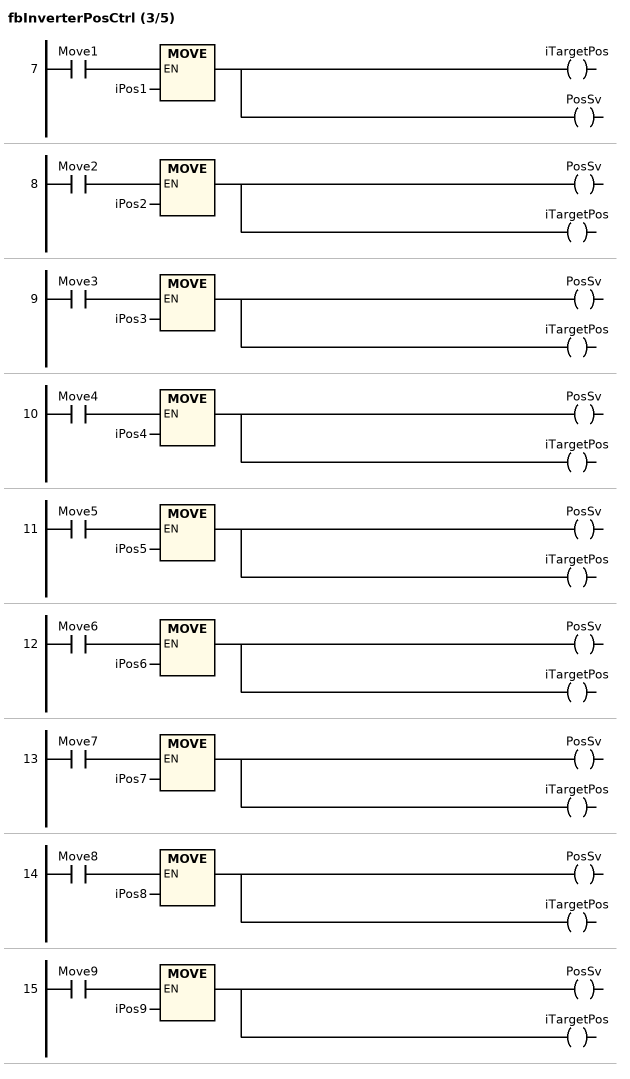
// NETWORK 7
IF Move1 THEN _w3 := iPos1; END_IF
iTargetPos := _w3;
PosSv := _w3;

// NETWORK 8
IF Move2 THEN _w4 := iPos2; END_IF
PosSv := _w4;
iTargetPos := _w4;

// NETWORK 9
IF Move3 THEN _w5 := iPos3; END_IF
PosSv := _w5;
iTargetPos := _w5;

// NETWORK 10
IF Move4 THEN _w6 := iPos4; END_IF
PosSv := _w6;
iTargetPos := _w6;

// NETWORK 11
IF Move5 THEN _w7 := iPos5; END_IF
PosSv := _w7;
iTargetPos := _w7;

// NETWORK 12
IF Move6 THEN _w8 := iPos6; END_IF
PosSv := _w8;
iTargetPos := _w8;

// NETWORK 13
IF Move7 THEN _w9 := iPos7; END_IF
PosSv := _w9;
iTargetPos := _w9;

// NETWORK 14
IF Move8 THEN _w10 := iPos8; END_IF
PosSv := _w10;
iTargetPos := _w10;

// NETWORK 15
IF Move9 THEN _w11 := iPos9; END_IF
PosSv := _w11;
iTargetPos := _w11;

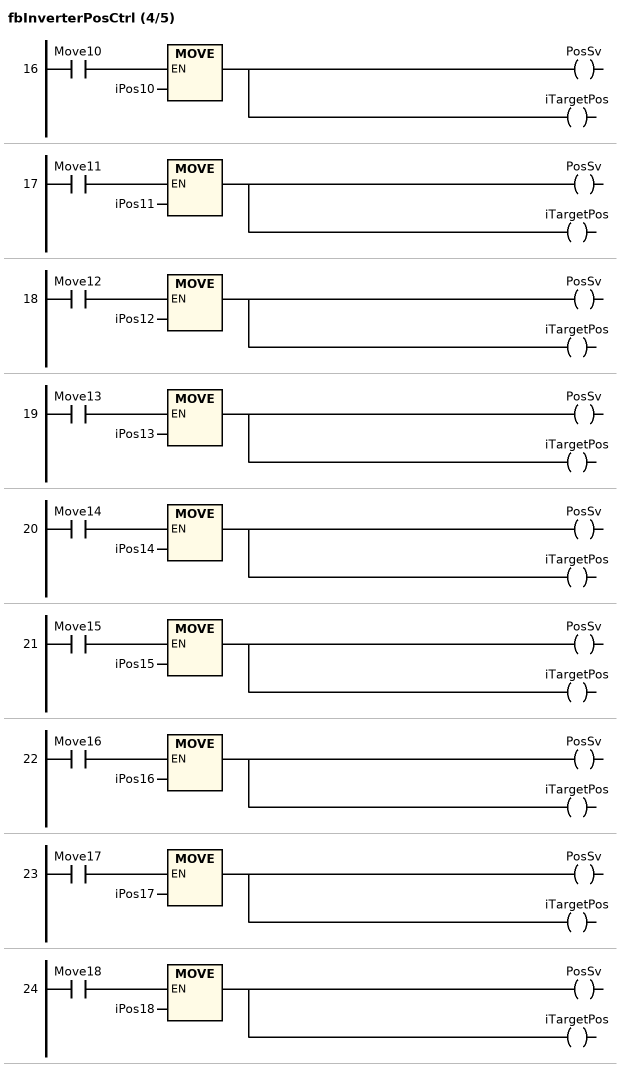
// NETWORK 16
IF Move10 THEN _w12 := iPos10; END_IF
PosSv := _w12;
iTargetPos := _w12;

// NETWORK 17
IF Move11 THEN _w13 := iPos11; END_IF
PosSv := _w13;
iTargetPos := _w13;

// NETWORK 18
IF Move12 THEN _w14 := iPos12; END_IF
PosSv := _w14;
iTargetPos := _w14;

// NETWORK 19
IF Move13 THEN _w15 := iPos13; END_IF
PosSv := _w15;
iTargetPos := _w15;

// NETWORK 20
IF Move14 THEN _w16 := iPos14; END_IF
PosSv := _w16;
iTargetPos := _w16;

// NETWORK 21
IF Move15 THEN _w17 := iPos15; END_IF
PosSv := _w17;
iTargetPos := _w17;

// NETWORK 22
IF Move16 THEN _w18 := iPos16; END_IF
PosSv := _w18;
iTargetPos := _w18;

// NETWORK 23
IF Move17 THEN _w19 := iPos17; END_IF
PosSv := _w19;
iTargetPos := _w19;

// NETWORK 24
IF Move18 THEN _w20 := iPos18; END_IF
PosSv := _w20;
iTargetPos := _w20;

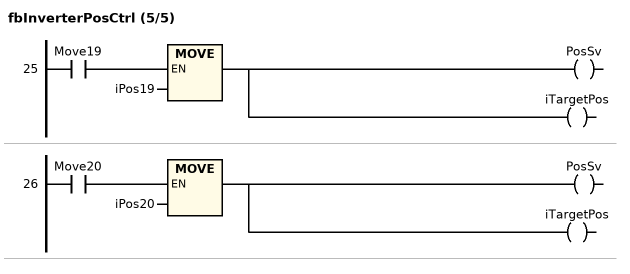
// NETWORK 25
IF Move19 THEN _w21 := iPos19; END_IF
PosSv := _w21;
iTargetPos := _w21;

// NETWORK 26
IF Move20 THEN _w22 := iPos20; END_IF
PosSv := _w22;
iTargetPos := _w22;

END_FUNCTION_BLOCK

// ---- FBs/B_JKS_CustomFB/fbArmCtrlFolder/fbInverterVertHome.TcPOU
FUNCTION_BLOCK fbInverterVertHome
VAR_INPUT
	bExecute	: BOOL;
	bEstop		: BOOL;
	bHomeFor	: BOOL;
	bHomeRev	: BOOL;
	bHomeSenser	: BOOL;
	bOTsensor1		: BOOL;
	bOTsensor2		: BOOL;
	bReset			: BOOL;
	i1stRPM			: INT;
	i2ndRPM			: INT;
	rInverterRatio		: REAL;
	EncoderRatio		: LREAL;

END_VAR
VAR_OUTPUT
	bDone		: BOOL;
	bBusy		: BOOL;
	bError		: BOOL;
	bMovForBit	: BOOL;
	bMovRevBit	: BOOL;
	bMovFor2ndBit	: BOOL;
	bMovRev2ndBit	: BOOL;
	bMovFor3rdBit	: BOOL;
	bMovRev3rdBit	: BOOL;
	lrActualPosReference	: LREAL;

END_VAR
VAR_IN_OUT

	iHomeHzout	: INT;
	Axis1		: axis_ref;

END_VAR
VAR
	MCRAP1: MC_ReadActualPosition;
	PowerRelay: TON;
	ArmMovActualPos: LREAL;
	RTRIG1: R_TRIG;
	Move2Home: BOOL;
	HomingStop: BOOL;
	Conv1: AM_InverterConversionHz;
	Conv2: AM_InverterConversionHz;
	CMP1: fbServoPosCmp;
	ArmReachHome: BOOL;
	Conv3: AM_InverterConversionHz;
	Conv4: AM_InverterConversionHz;
	MoveAwayHome: BOOL;
	Conv5: AM_InverterConversionHz;
	Conv6: AM_InverterConversionHz;
	HomingStep1: BOOL;
	MCSPOS1: MC_SetPosition;
	SetPosDone: BOOL;
	TON2: TON;
	T1: TON;
	T2: TON;
	HomeSensorTriggerBit: BOOL;
	HomingStep2: BOOL;
	OTstop: BOOL;
	TRIG1: R_TRIG;
	TRIG2: R_TRIG;
	RTRIG2: R_TRIG;
	i1stRPMTemp: INT;
	i2ndRPMTemp: INT;
	LrPosBeforeConvert: LREAL;
	TON10: TON;
END_VAR

VAR PERSISTENT

	HorzArmPos : LREAL;

END_VAR
VAR // added by the converter: edge detectors and wires of the graphical bodies
    _w1, _w2 : INT;
    _w3 : LREAL;
END_VAR

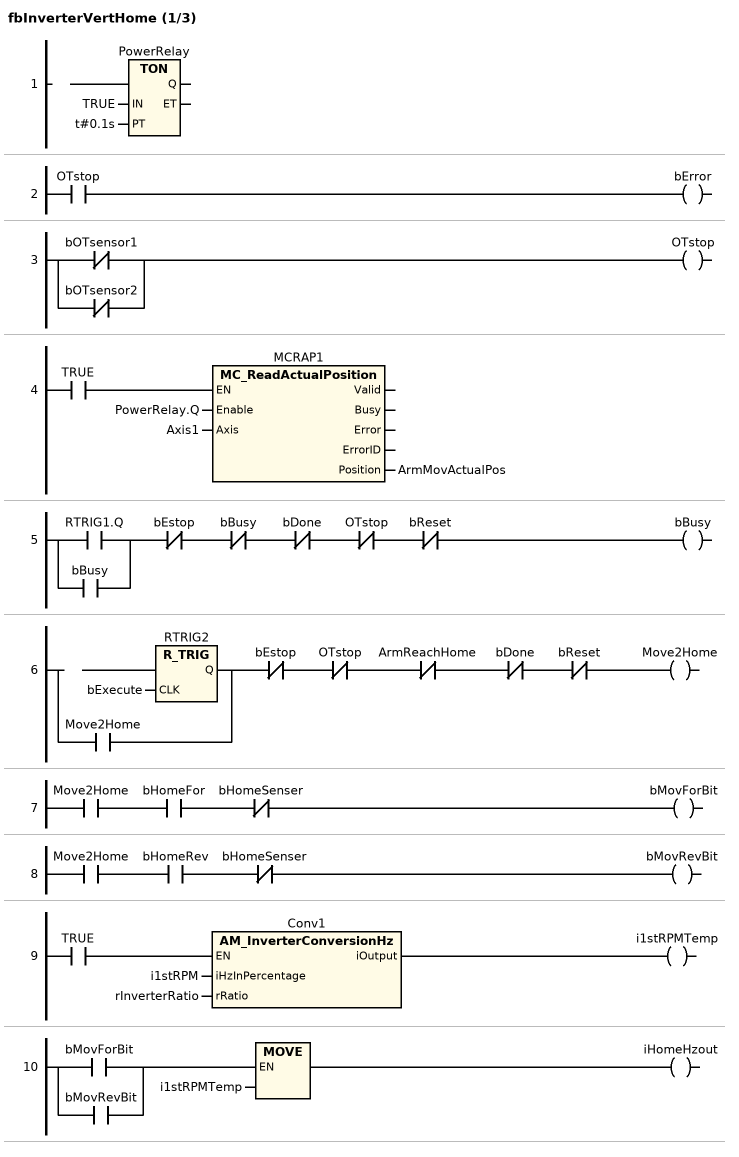
// NETWORK 1
PowerRelay(IN := TRUE, PT := t#0.1s); // TON

// NETWORK 2
bError := OTstop;

// NETWORK 3
OTstop := NOT bOTsensor1 OR NOT bOTsensor2;

// NETWORK 4
MCRAP1(Enable := PowerRelay.Q, Axis := Axis1, Position => ArmMovActualPos); // MC_ReadActualPosition

// NETWORK 5
bBusy := (RTRIG1.Q OR bBusy) AND NOT bEstop AND NOT bBusy AND NOT bDone AND NOT OTstop AND NOT bReset;

// NETWORK 6
RTRIG2(CLK := bExecute); // R_TRIG
Move2Home := (RTRIG2.Q OR Move2Home) AND NOT bEstop AND NOT OTstop AND NOT ArmReachHome AND NOT bDone AND NOT bReset;

// NETWORK 7
bMovForBit := Move2Home AND bHomeFor AND NOT bHomeSenser;

// NETWORK 8
bMovRevBit := Move2Home AND bHomeRev AND NOT bHomeSenser;

// NETWORK 9
Conv1(iHzInPercentage := i1stRPM, rRatio := rInverterRatio); // AM_InverterConversionHz
i1stRPMTemp := Conv1.iOutput;

// NETWORK 10
IF bMovForBit OR bMovRevBit THEN _w1 := i1stRPMTemp; END_IF
iHomeHzout := _w1;

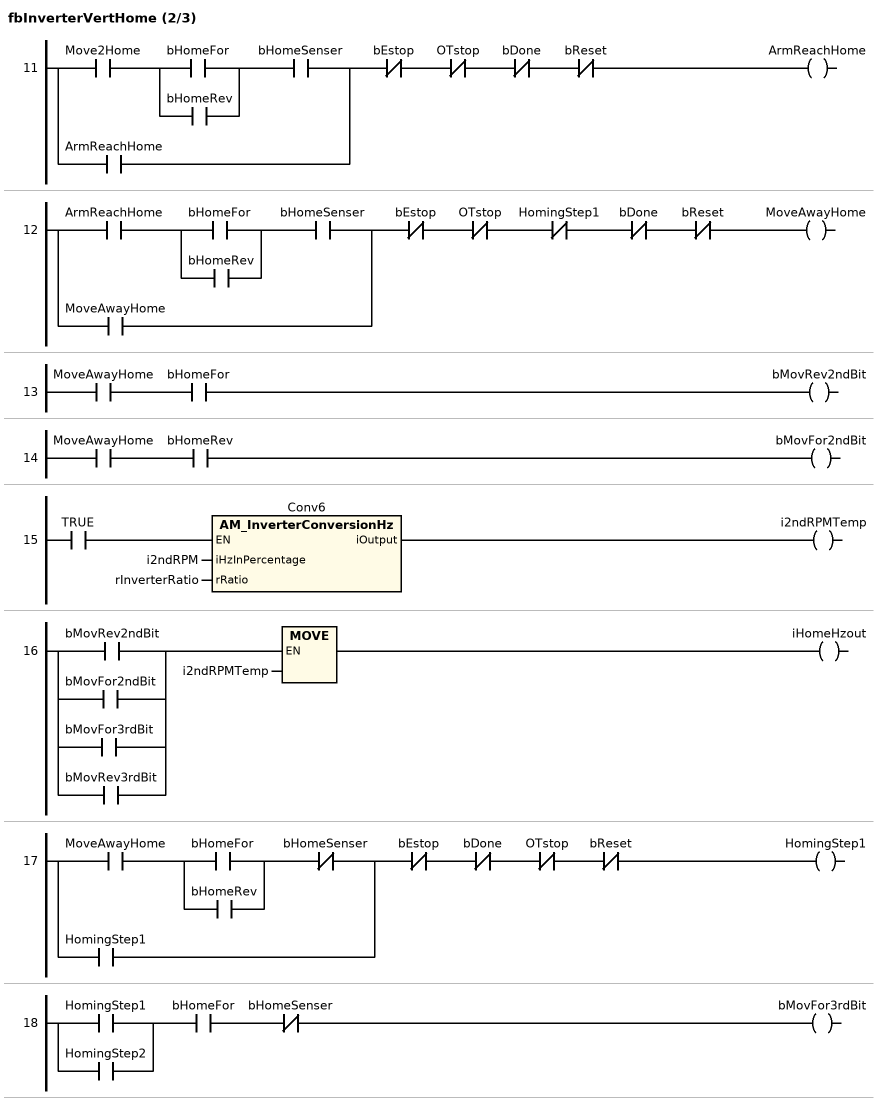
// NETWORK 11
ArmReachHome := ((Move2Home AND (bHomeFor OR bHomeRev)) AND bHomeSenser OR ArmReachHome) AND NOT bEstop AND NOT OTstop AND NOT bDone AND NOT bReset;

// NETWORK 12
MoveAwayHome := ((ArmReachHome AND (bHomeFor OR bHomeRev)) AND bHomeSenser OR MoveAwayHome) AND NOT bEstop AND NOT OTstop AND NOT HomingStep1 AND NOT bDone AND NOT bReset;

// NETWORK 13
bMovRev2ndBit := MoveAwayHome AND bHomeFor;

// NETWORK 14
bMovFor2ndBit := MoveAwayHome AND bHomeRev;

// NETWORK 15
Conv6(iHzInPercentage := i2ndRPM, rRatio := rInverterRatio); // AM_InverterConversionHz
i2ndRPMTemp := Conv6.iOutput;

// NETWORK 16
IF bMovRev2ndBit OR bMovFor2ndBit OR bMovFor3rdBit OR bMovRev3rdBit THEN _w2 := i2ndRPMTemp; END_IF
iHomeHzout := _w2;

// NETWORK 17
HomingStep1 := ((MoveAwayHome AND (bHomeFor OR bHomeRev)) AND NOT bHomeSenser OR HomingStep1) AND NOT bEstop AND NOT bDone AND NOT OTstop AND NOT bReset;

// NETWORK 18
bMovFor3rdBit := (HomingStep1 OR HomingStep2) AND bHomeFor AND NOT bHomeSenser;

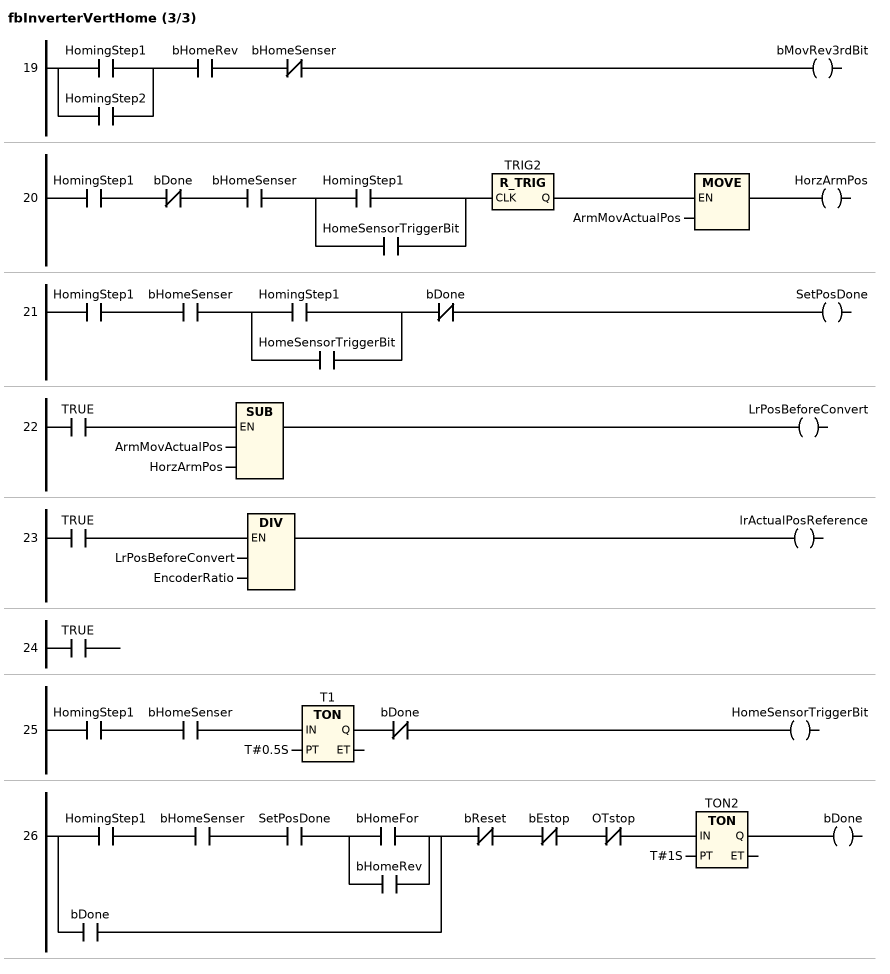
// NETWORK 19
bMovRev3rdBit := (HomingStep1 OR HomingStep2) AND bHomeRev AND NOT bHomeSenser;

// NETWORK 20
TRIG2(CLK := HomingStep1 AND NOT bDone AND bHomeSenser AND (HomingStep1 OR HomeSensorTriggerBit)); // R_TRIG
IF TRIG2.Q THEN _w3 := ArmMovActualPos; END_IF
HorzArmPos := _w3;

// NETWORK 21
SetPosDone := (HomingStep1 AND bHomeSenser AND (HomingStep1 OR HomeSensorTriggerBit)) AND NOT bDone;

// NETWORK 22
LrPosBeforeConvert := ArmMovActualPos - HorzArmPos;

// NETWORK 23
lrActualPosReference := LrPosBeforeConvert / EncoderRatio;

// NETWORK 24

// NETWORK 25
T1(IN := HomingStep1 AND bHomeSenser, PT := T#0.5S); // TON
HomeSensorTriggerBit := T1.Q AND NOT bDone;

// NETWORK 26
TON2(IN := (HomingStep1 AND bHomeSenser AND SetPosDone AND (bHomeFor OR bHomeRev) OR bDone) AND NOT bReset AND NOT bEstop AND NOT OTstop, PT := T#1S); // TON
bDone := TON2.Q;

END_FUNCTION_BLOCK

// ---- FBs/B_JKS_CustomFB/fbArmCtrlFolder/fbMotorHomingAxis.TcPOU
FUNCTION_BLOCK fbMotorHomingAxis
VAR_INPUT

	bEmergencyButton: BOOL;
	bHomingStart : BOOL ;
	lMoveVelo : LREAL;
	lMoveAcc : LREAL;
	lMoveDcc : LREAL;
	lMove2ndVelo : LREAL;
	lMove2ndAcc : LREAL;
	lMove2ndDcc : LREAL;
	bHomeSensor1 : BOOL;
	bOverTravelSensor1 : BOOL;
	bOverTravelSensor2 : BOOL;
	bReset : BOOL;
	tAlwaysHomeCompleteTimeDelay: TIME;
	tMCHomeStartDelay: TIME;


END_VAR

VAR_IN_OUT
	Axis1	: Axis_Ref;
	lrCurrentAxisPos : LREAL;
END_VAR

VAR_OUTPUT

	Home1Complete : BOOL;
END_VAR
VAR

	lrPosAxisAwayHome : LREAL := 9999;

	ArmStopBit: BOOL;
	HomingInterlocking: BOOL;
	ArmTouchHome: BOOL;
	bOverTravelSensor: BOOL;
	halt: MC_Halt;
	ArmHaltDone: BOOL;
	ArmBelowSensor: BOOL;
	bHomeSensor: BOOL;
	Move2home: BOOL;
	move1: MC_MoveRelative;
	moveBusy: BOOL;
	halt1: MC_Halt;
	ArmEstopDone: BOOL;
	Estop: BOOL;
	MoveAway: BOOL;
	move2: MC_MoveRelative;
	Timer1: TON;
	ArmAwayHome: BOOL;
	move3: MC_MoveRelative;
	AwayHomeBusy: BOOL;
	AwayHomeDone: BOOL;
	halt3: MC_Halt;
	AwayHaltDone: BOOL;
	HomingStart: BOOL;
	Delay: TON;
	Timer2: TON;
	home1: MC_Home;
	Home1Done: BOOL;
	Timer3: TON;
	step1: BOOL;
	Delay1: TON;
	HomeStartDIFU: R_TRIG;
	bPosError: BOOL;
	MCSP: MC_SetPosition;
	HomingStartEN_DIFU: R_TRIG;
	HomingStartFE: F_TRIG;
	PosErrorDIFU: R_TRIG;
	PosErrorTimer: TON;
	Home1Complete1: BOOL;
	Home1CompleteDIFU: R_TRIG;
	DON: TON;
END_VAR

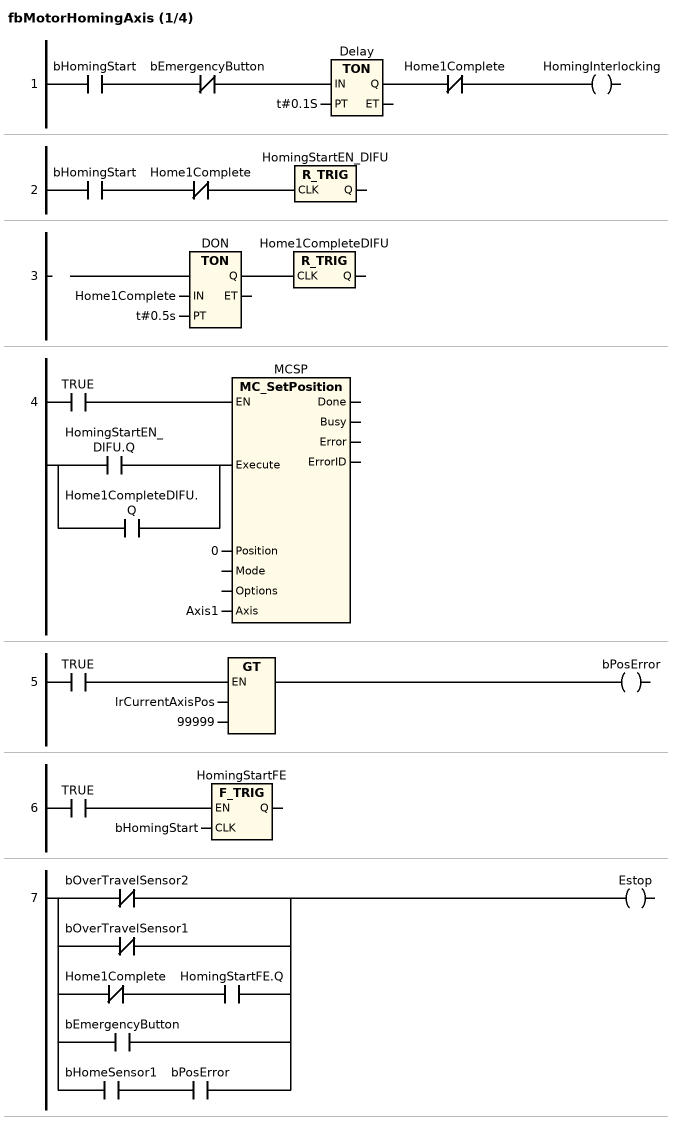
// NETWORK 1
Delay(IN := bHomingStart AND NOT bEmergencyButton, PT := t#0.1S); // TON
HomingInterlocking := Delay.Q AND NOT Home1Complete;

// NETWORK 2
HomingStartEN_DIFU(CLK := bHomingStart AND NOT Home1Complete); // R_TRIG

// NETWORK 3
DON(IN := Home1Complete, PT := t#0.5s); // TON
Home1CompleteDIFU(CLK := DON.Q); // R_TRIG

// NETWORK 4
MCSP(Execute := HomingStartEN_DIFU.Q OR Home1CompleteDIFU.Q, Position := 0, Axis := Axis1); // MC_SetPosition

// NETWORK 5
bPosError := lrCurrentAxisPos > 99999;

// NETWORK 6
HomingStartFE(CLK := bHomingStart); // F_TRIG

// NETWORK 7
Estop := NOT bOverTravelSensor2 OR NOT bOverTravelSensor1 OR NOT Home1Complete AND HomingStartFE.Q OR bEmergencyButton OR bHomeSensor1 AND bPosError;

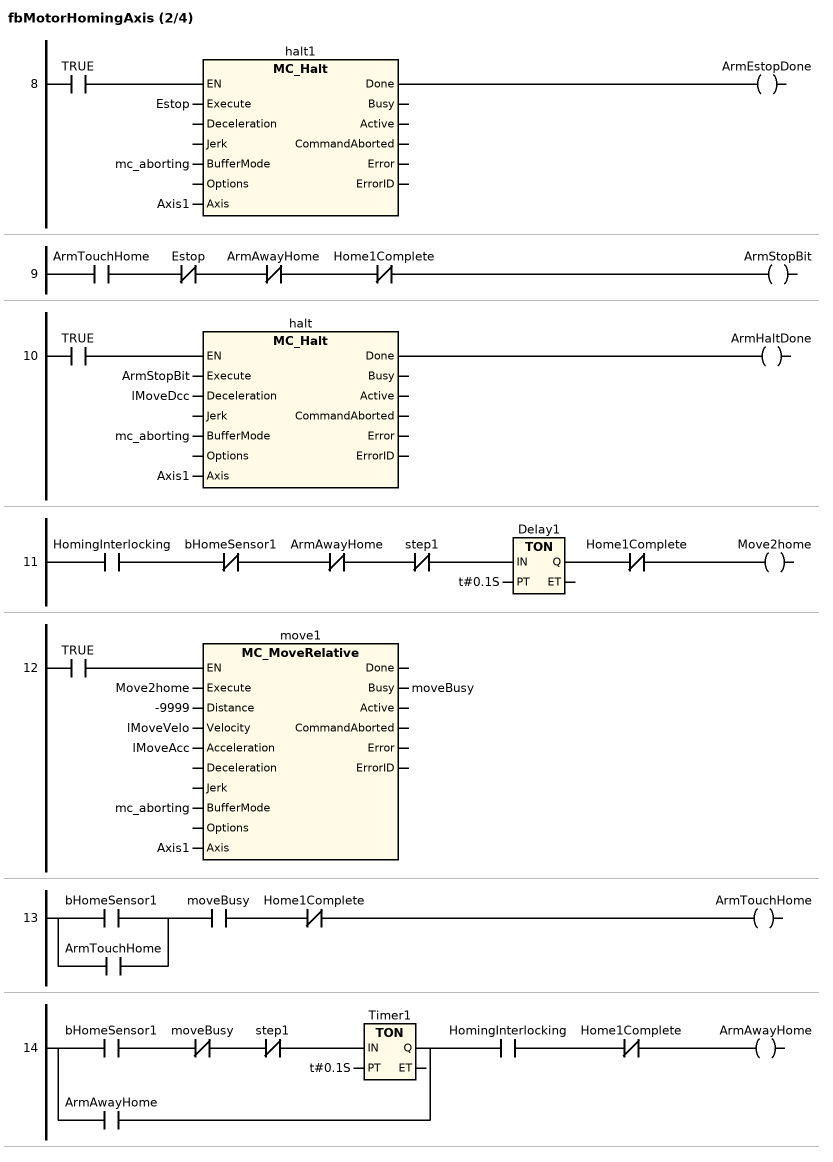
// NETWORK 8
halt1(Execute := Estop, BufferMode := mc_aborting, Axis := Axis1); // MC_Halt
ArmEstopDone := halt1.Done;

// NETWORK 9
ArmStopBit := ArmTouchHome AND NOT Estop AND NOT ArmAwayHome AND NOT Home1Complete;

// NETWORK 10
halt(Execute := ArmStopBit, Deceleration := lMoveDcc, BufferMode := mc_aborting, Axis := Axis1); // MC_Halt
ArmHaltDone := halt.Done;

// NETWORK 11
Delay1(IN := HomingInterlocking AND NOT bHomeSensor1 AND NOT ArmAwayHome AND NOT step1, PT := t#0.1S); // TON
Move2home := Delay1.Q AND NOT Home1Complete;

// NETWORK 12
move1(
    Execute := Move2home,
    Distance := -9999,
    Velocity := lMoveVelo,
    Acceleration := lMoveAcc,
    BufferMode := mc_aborting,
    Axis := Axis1,
    Busy => moveBusy); // MC_MoveRelative

// NETWORK 13
ArmTouchHome := (bHomeSensor1 OR ArmTouchHome) AND moveBusy AND NOT Home1Complete;

// NETWORK 14
Timer1(IN := bHomeSensor1 AND NOT moveBusy AND NOT step1, PT := t#0.1S); // TON
ArmAwayHome := (Timer1.Q OR ArmAwayHome) AND HomingInterlocking AND NOT Home1Complete;

